(* Logix 5000 project; controller Receptivo vendor 1 type 14 code 106 rev 30.11; software revision 30.00 *)

TASK HARDWARE_TESTING (periodic, rate 67.76 ms, priority 7, watchdog 500 ms) : SYSTEM_STATUS
TASK MainTask (continuous, watchdog 500 ms) : MainProgram, Pesaje, Manejo_Productos, Calculo_Produccion

MODULES
   Local : vendor 1 type 14 code 106 (Compact 0, rev 30.11)
      Printer_Code_2D : vendor 1421 type 43 code 1000 (Ethernet 192.168.105.118, rev 1.1, StandardDataDriven RPI 100 ms)
           Printer_Code_2D:O.RawParserData[15]   // SLASH
           Printer_Code_2D:O.RawParserData[18]   // SLASH
           Printer_Code_2D:O.RawParserData[22]   // espacio
           Printer_Code_2D:O.RawParserData[129]   // campo 12
           Printer_Code_2D:O.RawParserData[23]   // ESPACIO
           Printer_Code_2D:O.RawParserData[27]   // minutos
           Printer_Code_2D:O.RawParserData[28]   // espacio
           Printer_Code_2D:O.RawParserData[36]   // operador
           Printer_Code_2D:O.RawParserData[19]   // year
           Printer_Code_2D:O.RawParserData[20]   // year
           Printer_Code_2D:O.RawParserData[34]   // CLIMA
           Printer_Code_2D:O.RawParserData[3]   // campo 11
           Printer_Code_2D:O.RawParserData[105]   // espacio
           Printer_Code_2D:O.RawParserData[29]   // ESPACIO
           Printer_Code_2D:O.RawParserData[37]   // OPERADOR
           Printer_Code_2D:O.RawParserData[33]   // ESPACIO
           Printer_Code_2D:O.RawParserData[113]   // PESO REAL
           Printer_Code_2D:O.RawParserData[26]   // DOS PUNTOS
           Printer_Code_2D:O.RawParserData[8]   // field data
           Printer_Code_2D:O.RawParserData[35]   // ESPACIO
           Printer_Code_2D:O.RawParserData[21]   // year
           Printer_Code_2D:O.RawParserData[24]   // hora
           Printer_Code_2D:O.RawParserData[25]   // HORA
           Printer_Code_2D:O.RawParserData[30]   // lote
           Printer_Code_2D:O.RawParserData[31]   // lote
           Printer_Code_2D:O.RawParserData[32]   // LOTE
           Printer_Code_2D:O.RawParserData[13]   // dia
           Printer_Code_2D:O.RawParserData[14]   // DIA
           Printer_Code_2D:O.RawParserData[16]   // mes
           Printer_Code_2D:O.RawParserData[17]   // MES
           Printer_Code_2D:O.RawParserData[10]   // codigo QR
           Printer_Code_2D:O.RawParserData[112]   // ESPACIO
           Printer_Code_2D:O.RawParserData[116]   // ESPACIO
           Printer_Code_2D:O.RawParserData[91]   // CODIGO EAN14
           Printer_Code_2D:O.RawParserData[38]   // ESPACIO
           Printer_Code_2D:O.RawParserData[90]   // ESPACIO
           Printer_Code_2D:O.RawParserData[106]   // CODIGO QAD 6 CARACTERES
           Printer_Code_2D:O.RawParserData[124]   // separador
           Printer_Code_2D:O.RawParserData[11]   // codigo QR
           Printer_Code_2D:O.RawParserData[120]   // ESPACIO
           Printer_Code_2D:O.RawParserData[121]   // NUMERO DE CAJAS
           Printer_Code_2D:O.RawParserData[12]   // codigo qr
           Printer_Code_2D:O.RawParserData[117]   // peso teorico
           Printer_Code_2D:O.RawParserData[39]   // DESCRIPCION
           Printer_Code_2D:O.RawParserData[127]   // nuevo campo
           Printer_Code_2D:O.RawParserData[132]   // field 12 data
           Printer_Code_2D:O.RawParserData[125]   // Numero Estacion
      Hardy_Basculas : vendor 258 type 43 code 3 (Ethernet 192.168.105.216, rev 2.37, StandardDataDriven RPI 100 ms)
END_MODULES

TYPE APT :
STRUCT
   Cod_QAD : DINT;
   Peso : DINT;
   Cajas : DINT;
END_STRUCT
END_TYPE

TYPE Codigo_Barras :
STRUCT
   LEN : DINT;
   DATA : SINT[14];
END_STRUCT
END_TYPE

TYPE Consecutivo :
STRUCT
   Consec : STRING[3];
END_STRUCT
END_TYPE

TYPE Descripcion :
STRUCT
   LEN : DINT;
   DATA : SINT[45];
END_STRUCT
END_TYPE

TYPE Ethernet_Status :
STRUCT
   EntryStatus : DINT[256];
   ConnStatus : INT[256];
   ConnFault : BOOL[256];
END_STRUCT
END_TYPE

TYPE Hora_y_Fecha :
STRUCT
   year : DINT;
   Mes : DINT;
   Dia : DINT;
   Hora : DINT;
   Minuto : DINT;
   Segundo : DINT;
   Milisegundos : DINT;
END_STRUCT
END_TYPE

TYPE MajorFaultBits :
STRUCT
   B_reserved : BOOL;
   B_PowerLoss : BOOL;
   B_reserved1 : BOOL;
   B_IO : BOOL;
   B_InstructionExecution : BOOL;
   B_FaultHandler : BOOL;
   B_Watchdog : BOOL;
   B_Stack : BOOL;
   B_ModeChange : BOOL;
   B_reserved2 : BOOL;
   B_reserved3 : BOOL;
   B_Motion : BOOL;
   B_reserved4 : BOOL;
   B_reserved5 : BOOL;
   B_reserved6 : BOOL;
   B_reserved7 : BOOL;
END_STRUCT
END_TYPE

TYPE MinorFaultBits :
STRUCT
   B_reserved1 : BOOL;
   B_reserved2 : BOOL;
   B_reserved3 : BOOL;
   B_reserved4 : BOOL;
   B_InstructionExecution : BOOL;
   B_reserved5 : BOOL;
   B_Watchdog : BOOL;
   B_reserved7 : BOOL;
   B_reserved8 : BOOL;
   B_SerialPort : BOOL;
   B_Battery : BOOL;
   B_reserved11 : BOOL;
   B_reserved12 : BOOL;
   B_reserved13 : BOOL;
   B_reserved14 : BOOL;
   B_reserved15 : BOOL;
END_STRUCT
END_TYPE

TYPE QR :
STRUCT
   LEN : DINT;
   DATA : SINT[112];
END_STRUCT
END_TYPE

TYPE Revision_Peso :
STRUCT
   Date : Hora_y_Fecha;
   Peso_Real : REAL;
   Peso_Teorico : REAL;
   Codigo : STRING;
END_STRUCT
END_TYPE

TYPE UDT_CAJAS :
STRUCT
   No_Cajas : STRING[2];
END_STRUCT
END_TYPE

TYPE UDT_COLA :
STRUCT
   Fecha : Hora_y_Fecha;
   Lote : INT;
   Operador : SINT;
   Descripcion : STRING;
   EAN14 : STRING;
   QAD : STRING;
   Peso_Real : REAL;
   Peso_Teorico : REAL;
   No_Cajas : INT;
   Clima : SINT;
   Consec : DINT;
   Envase : DINT;
   Envases_x_Caja : DINT;
   Peso_Insumos_Caja : REAL;
   Densidad_Medida : REAL;
   Linea : SINT;
END_STRUCT
END_TYPE

TYPE UDT_Densidad :
STRUCT
   Densidad : REAL;
   Fecha : Hora_y_Fecha;
END_STRUCT
END_TYPE

TYPE UDT_EAN14 :   // campo nuero dos del codigo QR
STRUCT
   EAN14 : STRING;
END_STRUCT
END_TYPE

TYPE UDT_GENERAL :
STRUCT
   dd : STRING[2];
   mm : STRING[2];
   yy : STRING[4];
   hh : STRING[2];
   min : STRING[2];
   lote : STRING[3];
   clima : STRING;
   operador : STRING[2];
   Descripcion : STRING;
   EAN14 : STRING;
   QAD : STRING;
   Peso_Real : STRING[3];
   Peso_Teorico : STRING[3];
   No_Cajas : STRING[3];
   Linea : STRING;
END_STRUCT
END_TYPE

TYPE UDT_Inventario :
STRUCT
   Peso_Real : REAL;
   Peso_Teorico_Caja : REAL;
   Peso_Teorico_Estiba : REAL;
   Codigo_EAN : STRING;
   Codigo_QAD : STRING;
   Codigo_Gco : STRING;
   Descripcion : Descripcion;
   CajaXEstiba : INT;
   Lote : INT;
   Clima : SINT;
   Linea : SINT;
   Codigo_Aceite : DINT;
END_STRUCT
END_TYPE

TYPE UDT_Maestro :
STRUCT
   Peso_Real_Estiba : REAL;
   Peso_Teorico_Caja : REAL;
   Codigo_EAN : STRING;
   Codigo_QAD : STRING;
   Codigo_GCO : DINT;
   Descripcion : STRING;
   Cajas_X_Estiba : DINT;
   Clima : DINT;
   Codigo_Aceite : DINT;
   Envase : DINT;
   Envases_x_Caja : DINT;
END_STRUCT
END_TYPE

TYPE UDT_PESO_REAL :   // quinto campo del codigo QR
STRUCT
   Peso_Real : STRING[2];
END_STRUCT
END_TYPE

TYPE UDT_PESO_TEORICO :   // sexto campo del codigo QR
STRUCT
   Peso_Teorico : STRING[2];
END_STRUCT
END_TYPE

TYPE UDT_Productos :   // Base de datos de Productos
STRUCT
   Peso_Real : REAL;
   Peso_Teorico_Caja : REAL;
   Codigo_EAN : Codigo_Barras;
   Codigo_QAD : DINT;
   Codigo_GCO : DINT;
   Cajas_x_Estiba : DINT;
   Clima : DINT;
   Descripcion : Descripcion;
END_STRUCT
END_TYPE

TYPE UDT_QAD :   // campo tres del codigo QR
STRUCT
   Codigo : STRING;
END_STRUCT
END_TYPE

TYPE WPM_Status :
STRUCT
   ADC_Error : BOOL;
   Reserved1 : BOOL;
   Not_Connected : BOOL;
   Over_Range : BOOL;
   Reserved2 : BOOL;
   Reserved3 : BOOL;
   In_Motion : BOOL;
   Firmware_Update : BOOL;
   Missing_Sample : BOOL;
   Channel_Off : BOOL;
   Failed_To_Save_To_Memory : BOOL;
   Update_In_Progress : BOOL;
   Failed_To_Update : BOOL;
   Saving_To_Memory : BOOL;
   It_Test_In_Progress : BOOL;
   Parameter_ID_Not_Found : BOOL;
   dato1 : INT;
END_STRUCT
END_TYPE

VAR_GLOBAL   (* controller tags *)
   ACTIVE_SLOT : DINT[10];
   Actualiza1_Timer : TIMER := (PRE := 7000);
   Actualiza2_Timer : TIMER := (PRE := 9000);
   Actualiza3_Timer : TIMER := (PRE := 6000);
   Actualiza4_Timer : TIMER := (PRE := 6000);
   Actualiza_Reporte_1 : BOOL;
   Actualiza_Reporte_2 : BOOL;
   Actualiza_Reporte_3 : BOOL;
   Actualiza_Reporte_4 : BOOL;
   ando : DINT := -1073741824;
   Ano_Biciesto : INT := 2020;
   Autonegotiation_Fallo : BOOL;
   Autonegotiation_OK : BOOL := 1;
   Autonegotiation_Start : BOOL;
   AutoNegotiation_Status : SINT := 3;
   Bit_Medianoche : BOOL;
   bit_ptobar : BOOL;
   CAJAS_1 : DINT := 50;
   CAJAS_2 : DINT := 56;
   CAJAS_3 : DINT := 50;
   CAJAS_4 : DINT := 48;
   Cajas_Aux : DINT;
   Cajas_Aux_Scanner : STRING;
   Cajas_Calculadas_Estacion_1 : REAL := -1.3294798;
   Cajas_Calculadas_Estacion_2 : REAL := -2.8708134;
   Cajas_Calculadas_Estacion_3 : REAL;
   Cajas_Calculadas_Estacion_4 : REAL := -1.4041514;
   Cajas_CalculadasG_Estacion_1 : REAL := 49.59538;
   Cajas_CalculadasG_Estacion_2 : REAL := 52.440193;
   Cajas_CalculadasG_Estacion_3 : REAL := 3.0057805;
   Cajas_CalculadasG_Estacion_4 : REAL := 48.046402;
   Calendario : Hora_y_Fecha := (year := 2021, Mes := 5, Dia := 28, Hora := 16, Minuto := 19, Segundo := 32, Milisegundos := 517635);
   Cant_total : SINT := 50;
   Cantidad_de_Productos : DINT := 117;
   CERO : DINT;
   CEROS : SINT;
   CHASSIS_LAST : DINT := 1;
   CINCO : SINT := 5;
   Clima_1 : DINT;
   Clima_2 : DINT;
   Clima_3 : DINT;
   Clima_4 : DINT;
   CLOCK : DINT[7] := ([0] := 2021, [1] := 5, [2] := 28, [3] := 16, [4] := 19, [5] := 33, [6] := 245632);
   codigo_capturado_1 : BOOL;
   codigo_capturado_2 : BOOL;
   codigo_capturado_3 : BOOL;
   codigo_capturado_4 : BOOL;
   Codigo_Encontrado : BOOL := 1;
   Codigo_QAD2_Espacios : DINT := 112;
   Cola_Densidad_Bidon_Ayer : REAL[50];
   Cola_Densidad_Bidon_Fecha_Ayer : Hora_y_Fecha[50];
   Cola_Densidad_Bidones : REAL[50];
   Cola_Densidad_Bidones_Fecha : Hora_y_Fecha[50];
   Cola_Densidad_Bidones_Fecha_Ayer : Hora_y_Fecha[50];
   Cola_Densidad_Elmar : REAL[50];
   Cola_Densidad_Elmar_Ayer : REAL[50];
   Cola_Densidad_Elmar_Fecha : Hora_y_Fecha[50];
   Cola_Densidad_Elmar_Fecha_Ayer : Hora_y_Fecha[50];
   Cola_Densidad_Fogg1 : REAL[50];
   Cola_Densidad_Fogg1_Ayer : REAL[50];
   Cola_Densidad_fogg1_Fecha : Hora_y_Fecha[50];
   Cola_Densidad_fogg1_Fecha_Ayer : Hora_y_Fecha[50];
   Cola_Densidad_Fogg2 : REAL[50];
   Cola_Densidad_Fogg2_Ayer : REAL[50];
   Cola_Densidad_fogg2_Fecha : Hora_y_Fecha[50];
   Cola_Densidad_fogg2_Fecha_Ayer : Hora_y_Fecha[50];
   Cola_Densidad_Karat : REAL[50];
   Cola_Densidad_Karat_Ayer : REAL[50];
   Cola_Densidad_Karat_Fecha : Hora_y_Fecha[50];
   Cola_Densidad_Karat_Fecha_Ayer : Hora_y_Fecha[50];
   Cola_Estacion_1 : UDT_COLA[100];
   Cola_Estacion_1_A : UDT_COLA[100];
   Cola_Estacion_2 : UDT_COLA[100] := ([0].Fecha.year := 2021, [0].Fecha.Mes := 5, [0].Fecha.Dia := 28, [0].Fecha.Hora := 11, [0].Fecha.Minuto := 23, [0].Fecha.Segundo := 35, [0].Fecha.Milisegundos := 472457, [0].Lote := 148, [0].Operador := 5, [0].Descripcion := 'Alegria Caja 12 x 900 cm3  - Costa', [0].EAN14 := '17702161409646', [0].QAD := '600620', [0].Peso_Real := 589.0, [0].Peso_Teorico := 585.0, [0].No_Cajas := 56, [0].Consec := 31, [0].Envase := 900, [0].Envases_x_Caja := 12, [0].Densidad_Medida := 0.9152, [0].Linea := 1, [1].Fecha.year := 2021, [1].Fecha.Mes := 5, [1].Fecha.Dia := 28, [1].Fecha.Hora := 11, [1].Fecha.Minuto := 26, [1].Fecha.Segundo := 22, [1].Fecha.Milisegundos := 21267, [1].Lote := 148, [1].Operador := 5, [1].Descripcion := 'Alegria Caja 12 x 900 cm3  - Costa', [1].EAN14 := '17702161409646', [1].QAD := '600620', [1].Peso_Real := 590.0, [1].Peso_Teorico := 585.0, [1].No_Cajas := 56, [1].Consec := 32, [1].Envase := 900, [1].Envases_x_Caja := 12, [1].Densidad_Medida := 0.9152, [1].Linea := 1, [2].Fecha.year := 2021, [2].Fecha.Mes := 5, [2].Fecha.Dia := 28, [2].Fecha.Hora := 11, [2].Fecha.Minuto := 29, [2].Fecha.Segundo := 36, [2].Fecha.Milisegundos := 993294, [2].Lote := 148, [2].Operador := 5, [2].Descripcion := 'Alegria Caja 12 x 900 cm3  - Costa', [2].EAN14 := '17702161409646', [2].QAD := '600620', [2].Peso_Real := 584.0, [2].Peso_Teorico := 585.0, [2].No_Cajas := 56, [2].Consec := 33, [2].Envase := 900, [2].Envases_x_Caja := 12, [2].Densidad_Medida := 0.9152, [2].Linea := 1,
        [3].Fecha.year := 2021, [3].Fecha.Mes := 5, [3].Fecha.Dia := 28, [3].Fecha.Hora := 11, [3].Fecha.Minuto := 32, [3].Fecha.Segundo := 47, [3].Fecha.Milisegundos := 567933, [3].Lote := 148, [3].Operador := 5, [3].Descripcion := 'Alegria Caja 12 x 900 cm3  - Costa', [3].EAN14 := '17702161409646', [3].QAD := '600620', [3].Peso_Real := 589.0, [3].Peso_Teorico := 585.0, [3].No_Cajas := 56, [3].Consec := 34, [3].Envase := 900, [3].Envases_x_Caja := 12, [3].Densidad_Medida := 0.9152, [3].Linea := 1, [4].Fecha.year := 2021, [4].Fecha.Mes := 5, [4].Fecha.Dia := 28, [4].Fecha.Hora := 11, [4].Fecha.Minuto := 35, [4].Fecha.Segundo := 25, [4].Fecha.Milisegundos := 115498, [4].Lote := 148, [4].Operador := 5, [4].Descripcion := 'Alegria Caja 12 x 900 cm3  - Costa', [4].EAN14 := '17702161409646', [4].QAD := '600620', [4].Peso_Real := 590.0, [4].Peso_Teorico := 585.0, [4].No_Cajas := 56, [4].Consec := 35, [4].Envase := 900, [4].Envases_x_Caja := 12, [4].Densidad_Medida := 0.9152, [4].Linea := 1, [5].Fecha.year := 2021, [5].Fecha.Mes := 5, [5].Fecha.Dia := 28, [5].Fecha.Hora := 11, [5].Fecha.Minuto := 38, [5].Fecha.Segundo := 2, [5].Fecha.Milisegundos := 738210, [5].Lote := 148, [5].Operador := 5, [5].Descripcion := 'Alegria Caja 12 x 900 cm3  - Costa', [5].EAN14 := '17702161409646', [5].QAD := '600620', [5].Peso_Real := 589.0, [5].Peso_Teorico := 585.0, [5].No_Cajas := 56, [5].Consec := 36, [5].Envase := 900, [5].Envases_x_Caja := 12, [5].Densidad_Medida := 0.9152, [5].Linea := 1,
        [6].Fecha.year := 2021, [6].Fecha.Mes := 5, [6].Fecha.Dia := 28, [6].Fecha.Hora := 11, [6].Fecha.Minuto := 40, [6].Fecha.Segundo := 46, [6].Fecha.Milisegundos := 866704, [6].Lote := 148, [6].Operador := 5, [6].Descripcion := 'Alegria Caja 12 x 900 cm3  - Costa', [6].EAN14 := '17702161409646', [6].QAD := '600620', [6].Peso_Real := 590.0, [6].Peso_Teorico := 585.0, [6].No_Cajas := 56, [6].Consec := 38, [6].Envase := 900, [6].Envases_x_Caja := 12, [6].Densidad_Medida := 0.9152, [6].Linea := 1, [7].Fecha.year := 2021, [7].Fecha.Mes := 5, [7].Fecha.Dia := 28, [7].Fecha.Hora := 11, [7].Fecha.Minuto := 44, [7].Fecha.Segundo := 7, [7].Fecha.Milisegundos := 219454, [7].Lote := 148, [7].Operador := 5, [7].Descripcion := 'Alegria Caja 12 x 900 cm3  - Costa', [7].EAN14 := '17702161409646', [7].QAD := '600620', [7].Peso_Real := 590.0, [7].Peso_Teorico := 585.0, [7].No_Cajas := 56, [7].Consec := 40, [7].Envase := 900, [7].Envases_x_Caja := 12, [7].Densidad_Medida := 0.9152, [7].Linea := 1, [8].Fecha.year := 2021, [8].Fecha.Mes := 5, [8].Fecha.Dia := 28, [8].Fecha.Hora := 11, [8].Fecha.Minuto := 46, [8].Fecha.Segundo := 55, [8].Fecha.Milisegundos := 872733, [8].Lote := 148, [8].Operador := 5, [8].Descripcion := 'Alegria Caja 12 x 900 cm3  - Costa', [8].EAN14 := '17702161409646', [8].QAD := '600620', [8].Peso_Real := 590.0, [8].Peso_Teorico := 585.0, [8].No_Cajas := 56, [8].Consec := 41, [8].Envase := 900, [8].Envases_x_Caja := 12, [8].Densidad_Medida := 0.9152, [8].Linea := 1,
        [9].Fecha.year := 2021, [9].Fecha.Mes := 5, [9].Fecha.Dia := 28, [9].Fecha.Hora := 11, [9].Fecha.Minuto := 49, [9].Fecha.Segundo := 6, [9].Fecha.Milisegundos := 938412, [9].Lote := 148, [9].Operador := 5, [9].Descripcion := 'Alegria Caja 12 x 900 cm3  - Costa', [9].EAN14 := '17702161409646', [9].QAD := '600620', [9].Peso_Real := 590.0, [9].Peso_Teorico := 585.0, [9].No_Cajas := 56, [9].Consec := 43, [9].Envase := 900, [9].Envases_x_Caja := 12, [9].Densidad_Medida := 0.9152, [9].Linea := 1, [10].Fecha.year := 2021, [10].Fecha.Mes := 5, [10].Fecha.Dia := 28, [10].Fecha.Hora := 11, [10].Fecha.Minuto := 51, [10].Fecha.Segundo := 47, [10].Fecha.Milisegundos := 512506, [10].Lote := 148, [10].Operador := 5, [10].Descripcion := 'Alegria Caja 12 x 900 cm3  - Costa', [10].EAN14 := '17702161409646', [10].QAD := '600620', [10].Peso_Real := 590.0, [10].Peso_Teorico := 585.0, [10].No_Cajas := 56, [10].Consec := 44, [10].Envase := 900, [10].Envases_x_Caja := 12, [10].Densidad_Medida := 0.9152, [10].Linea := 1, [11].Fecha.year := 2021, [11].Fecha.Mes := 5, [11].Fecha.Dia := 28, [11].Fecha.Hora := 11, [11].Fecha.Minuto := 54, [11].Fecha.Segundo := 6, [11].Fecha.Milisegundos := 98780, [11].Lote := 148, [11].Operador := 5, [11].Descripcion := 'Alegria Caja 12 x 900 cm3  - Costa', [11].EAN14 := '17702161409646', [11].QAD := '600620', [11].Peso_Real := 590.0, [11].Peso_Teorico := 585.0, [11].No_Cajas := 56, [11].Consec := 45, [11].Envase := 900, [11].Envases_x_Caja := 12, [11].Densidad_Medida := 0.9152, [11].Linea := 1,
        [12].Fecha.year := 2021, [12].Fecha.Mes := 5, [12].Fecha.Dia := 28, [12].Fecha.Hora := 11, [12].Fecha.Minuto := 56, [12].Fecha.Segundo := 16, [12].Fecha.Milisegundos := 868293, [12].Lote := 148, [12].Operador := 5, [12].Descripcion := 'Alegria Caja 12 x 900 cm3  - Costa', [12].EAN14 := '17702161409646', [12].QAD := '600620', [12].Peso_Real := 591.0, [12].Peso_Teorico := 585.0, [12].No_Cajas := 56, [12].Consec := 47, [12].Envase := 900, [12].Envases_x_Caja := 12, [12].Densidad_Medida := 0.9152, [12].Linea := 1, [13].Fecha.year := 2021, [13].Fecha.Mes := 5, [13].Fecha.Dia := 28, [13].Fecha.Hora := 11, [13].Fecha.Minuto := 58, [13].Fecha.Segundo := 33, [13].Fecha.Milisegundos := 275353, [13].Lote := 148, [13].Operador := 5, [13].Descripcion := 'Alegria Caja 12 x 900 cm3  - Costa', [13].EAN14 := '17702161409646', [13].QAD := '600620', [13].Peso_Real := 591.0, [13].Peso_Teorico := 585.0, [13].No_Cajas := 56, [13].Consec := 48, [13].Envase := 900, [13].Envases_x_Caja := 12, [13].Densidad_Medida := 0.9152, [13].Linea := 1, [14].Fecha.year := 2021, [14].Fecha.Mes := 5, [14].Fecha.Dia := 28, [14].Fecha.Hora := 12, [14].Fecha.Segundo := 51, [14].Fecha.Milisegundos := 241323, [14].Lote := 148, [14].Operador := 5, [14].Descripcion := 'Alegria Caja 12 x 900 cm3  - Costa', [14].EAN14 := '17702161409646', [14].QAD := '600620', [14].Peso_Real := 590.0, [14].Peso_Teorico := 585.0, [14].No_Cajas := 56, [14].Consec := 49, [14].Envase := 900, [14].Envases_x_Caja := 12, [14].Densidad_Medida := 0.9152, [14].Linea := 1, [15].Fecha.year := 2021,
        [15].Fecha.Mes := 5, [15].Fecha.Dia := 28, [15].Fecha.Hora := 12, [15].Fecha.Minuto := 3, [15].Fecha.Segundo := 25, [15].Fecha.Milisegundos := 977302, [15].Lote := 148, [15].Operador := 5, [15].Descripcion := 'Alegria Caja 12 x 900 cm3  - Costa', [15].EAN14 := '17702161409646', [15].QAD := '600620', [15].Peso_Real := 589.0, [15].Peso_Teorico := 585.0, [15].No_Cajas := 56, [15].Consec := 50, [15].Envase := 900, [15].Envases_x_Caja := 12, [15].Densidad_Medida := 0.9152, [15].Linea := 1, [16].Fecha.year := 2021, [16].Fecha.Mes := 5, [16].Fecha.Dia := 28, [16].Fecha.Hora := 12, [16].Fecha.Minuto := 5, [16].Fecha.Segundo := 59, [16].Fecha.Milisegundos := 211755, [16].Lote := 148, [16].Operador := 5, [16].Descripcion := 'Alegria Caja 12 x 900 cm3  - Costa', [16].EAN14 := '17702161409646', [16].QAD := '600620', [16].Peso_Real := 589.0, [16].Peso_Teorico := 585.0, [16].No_Cajas := 56, [16].Consec := 51, [16].Envase := 900, [16].Envases_x_Caja := 12, [16].Densidad_Medida := 0.9152, [16].Linea := 1, [17].Fecha.year := 2021, [17].Fecha.Mes := 5, [17].Fecha.Dia := 28, [17].Fecha.Hora := 12, [17].Fecha.Minuto := 8, [17].Fecha.Segundo := 18, [17].Fecha.Milisegundos := 641820, [17].Lote := 148, [17].Operador := 5, [17].Descripcion := 'Alegria Caja 12 x 900 cm3  - Costa', [17].EAN14 := '17702161409646', [17].QAD := '600620', [17].Peso_Real := 589.0, [17].Peso_Teorico := 585.0, [17].No_Cajas := 56, [17].Consec := 52, [17].Envase := 900, [17].Envases_x_Caja := 12, [17].Densidad_Medida := 0.9152, [17].Linea := 1, [18].Fecha.year := 2021,
        [18].Fecha.Mes := 5, [18].Fecha.Dia := 28, [18].Fecha.Hora := 12, [18].Fecha.Minuto := 10, [18].Fecha.Segundo := 49, [18].Fecha.Milisegundos := 898961, [18].Lote := 148, [18].Operador := 5, [18].Descripcion := 'Alegria Caja 12 x 900 cm3  - Costa', [18].EAN14 := '17702161409646', [18].QAD := '600620', [18].Peso_Real := 589.0, [18].Peso_Teorico := 585.0, [18].No_Cajas := 56, [18].Consec := 53, [18].Envase := 900, [18].Envases_x_Caja := 12, [18].Densidad_Medida := 0.9152, [18].Linea := 1, [19].Fecha.year := 2021, [19].Fecha.Mes := 5, [19].Fecha.Dia := 28, [19].Fecha.Hora := 12, [19].Fecha.Minuto := 12, [19].Fecha.Segundo := 58, [19].Fecha.Milisegundos := 826984, [19].Lote := 148, [19].Operador := 5, [19].Descripcion := 'Alegria Caja 12 x 900 cm3  - Costa', [19].EAN14 := '17702161409646', [19].QAD := '600620', [19].Peso_Real := 589.0, [19].Peso_Teorico := 585.0, [19].No_Cajas := 56, [19].Consec := 54, [19].Envase := 900, [19].Envases_x_Caja := 12, [19].Densidad_Medida := 0.9152, [19].Linea := 1, [20].Fecha.year := 2021, [20].Fecha.Mes := 5, [20].Fecha.Dia := 28, [20].Fecha.Hora := 12, [20].Fecha.Minuto := 15, [20].Fecha.Segundo := 28, [20].Fecha.Milisegundos := 245825, [20].Lote := 148, [20].Operador := 5, [20].Descripcion := 'Alegria Caja 12 x 900 cm3  - Costa', [20].EAN14 := '17702161409646', [20].QAD := '600620', [20].Peso_Real := 588.0, [20].Peso_Teorico := 585.0, [20].No_Cajas := 56, [20].Consec := 55, [20].Envase := 900, [20].Envases_x_Caja := 12, [20].Densidad_Medida := 0.9152, [20].Linea := 1, [21].Fecha.year := 2021,
        [21].Fecha.Mes := 5, [21].Fecha.Dia := 28, [21].Fecha.Hora := 12, [21].Fecha.Minuto := 17, [21].Fecha.Segundo := 41, [21].Fecha.Milisegundos := 646158, [21].Lote := 148, [21].Operador := 5, [21].Descripcion := 'Alegria Caja 12 x 900 cm3  - Costa', [21].EAN14 := '17702161409646', [21].QAD := '600620', [21].Peso_Real := 589.0, [21].Peso_Teorico := 585.0, [21].No_Cajas := 56, [21].Consec := 56, [21].Envase := 900, [21].Envases_x_Caja := 12, [21].Densidad_Medida := 0.9152, [21].Linea := 1, [22].Fecha.year := 2021, [22].Fecha.Mes := 5, [22].Fecha.Dia := 28, [22].Fecha.Hora := 12, [22].Fecha.Minuto := 20, [22].Fecha.Segundo := 40, [22].Fecha.Milisegundos := 210367, [22].Lote := 148, [22].Operador := 5, [22].Descripcion := 'Alegria Caja 12 x 900 cm3  - Costa', [22].EAN14 := '17702161409646', [22].QAD := '600620', [22].Peso_Real := 588.0, [22].Peso_Teorico := 585.0, [22].No_Cajas := 56, [22].Consec := 57, [22].Envase := 900, [22].Envases_x_Caja := 12, [22].Densidad_Medida := 0.9152, [22].Linea := 1, [23].Fecha.year := 2021, [23].Fecha.Mes := 5, [23].Fecha.Dia := 28, [23].Fecha.Hora := 12, [23].Fecha.Minuto := 22, [23].Fecha.Segundo := 35, [23].Fecha.Milisegundos := 762553, [23].Lote := 148, [23].Operador := 5, [23].Descripcion := 'Alegria Caja 12 x 900 cm3  - Costa', [23].EAN14 := '17702161409646', [23].QAD := '600620', [23].Peso_Real := 590.0, [23].Peso_Teorico := 585.0, [23].No_Cajas := 56, [23].Consec := 58, [23].Envase := 900, [23].Envases_x_Caja := 12, [23].Densidad_Medida := 0.9152, [23].Linea := 1, [24].Fecha.year := 2021,
        [24].Fecha.Mes := 5, [24].Fecha.Dia := 28, [24].Fecha.Hora := 12, [24].Fecha.Minuto := 29, [24].Fecha.Segundo := 23, [24].Fecha.Milisegundos := 722342, [24].Lote := 148, [24].Operador := 5, [24].Descripcion := 'Alegria Caja 12 x 900 cm3  - Costa', [24].EAN14 := '17702161409646', [24].QAD := '600620', [24].Peso_Real := 587.0, [24].Peso_Teorico := 585.0, [24].No_Cajas := 56, [24].Consec := 59, [24].Envase := 900, [24].Envases_x_Caja := 12, [24].Densidad_Medida := 0.9152, [24].Linea := 1, [25].Fecha.year := 2021, [25].Fecha.Mes := 5, [25].Fecha.Dia := 28, [25].Fecha.Hora := 12, [25].Fecha.Minuto := 36, [25].Fecha.Segundo := 23, [25].Fecha.Milisegundos := 316720, [25].Lote := 148, [25].Operador := 5, [25].Descripcion := 'Alegria Caja 12 x 900 cm3  - Costa', [25].EAN14 := '17702161409646', [25].QAD := '600620', [25].Peso_Real := 586.0, [25].Peso_Teorico := 585.0, [25].No_Cajas := 56, [25].Consec := 60, [25].Envase := 900, [25].Envases_x_Caja := 12, [25].Densidad_Medida := 0.9152, [25].Linea := 1, [26].Fecha.year := 2021, [26].Fecha.Mes := 5, [26].Fecha.Dia := 28, [26].Fecha.Hora := 12, [26].Fecha.Minuto := 38, [26].Fecha.Segundo := 23, [26].Fecha.Milisegundos := 44403, [26].Lote := 148, [26].Operador := 5, [26].Descripcion := 'Alegria Caja 12 x 900 cm3  - Costa', [26].EAN14 := '17702161409646', [26].QAD := '600620', [26].Peso_Real := 579.0, [26].Peso_Teorico := 585.0, [26].No_Cajas := 56, [26].Consec := 62, [26].Envase := 900, [26].Envases_x_Caja := 12, [26].Densidad_Medida := 0.9152, [26].Linea := 1, [27].Fecha.year := 2021,
        [27].Fecha.Mes := 5, [27].Fecha.Dia := 28, [27].Fecha.Hora := 12, [27].Fecha.Minuto := 47, [27].Fecha.Segundo := 26, [27].Fecha.Milisegundos := 654204, [27].Lote := 148, [27].Operador := 5, [27].Descripcion := 'Alegria Caja 12 x 900 cm3  - Costa', [27].EAN14 := '17702161409646', [27].QAD := '600620', [27].Peso_Real := 578.0, [27].Peso_Teorico := 585.0, [27].No_Cajas := 56, [27].Consec := 63, [27].Envase := 900, [27].Envases_x_Caja := 12, [27].Densidad_Medida := 0.9152, [27].Linea := 1, [28].Fecha.year := 2021, [28].Fecha.Mes := 5, [28].Fecha.Dia := 28, [28].Fecha.Hora := 12, [28].Fecha.Minuto := 50, [28].Fecha.Segundo := 58, [28].Fecha.Milisegundos := 76476, [28].Lote := 148, [28].Operador := 5, [28].Descripcion := 'Alegria Caja 12 x 900 cm3  - Costa', [28].EAN14 := '17702161409646', [28].QAD := '600620', [28].Peso_Real := 602.0, [28].Peso_Teorico := 585.0, [28].No_Cajas := 56, [28].Consec := 65, [28].Envase := 900, [28].Envases_x_Caja := 12, [28].Densidad_Medida := 0.9152, [28].Linea := 1, [29].Fecha.year := 2021, [29].Fecha.Mes := 5, [29].Fecha.Dia := 28, [29].Fecha.Hora := 12, [29].Fecha.Minuto := 53, [29].Fecha.Segundo := 51, [29].Fecha.Milisegundos := 99875, [29].Lote := 148, [29].Operador := 5, [29].Descripcion := 'Alegria Caja 12 x 900 cm3  - Costa', [29].EAN14 := '17702161409646', [29].QAD := '600620', [29].Peso_Real := 592.0, [29].Peso_Teorico := 585.0, [29].No_Cajas := 56, [29].Consec := 67, [29].Envase := 900, [29].Envases_x_Caja := 12, [29].Densidad_Medida := 0.9152, [29].Linea := 1, [30].Fecha.year := 2021,
        [30].Fecha.Mes := 5, [30].Fecha.Dia := 28, [30].Fecha.Hora := 13, [30].Fecha.Minuto := 3, [30].Fecha.Segundo := 33, [30].Fecha.Milisegundos := 200046, [30].Lote := 148, [30].Operador := 5, [30].Descripcion := 'Alegria Caja 12 x 900 cm3  - Costa', [30].EAN14 := '17702161409646', [30].QAD := '600620', [30].Peso_Real := 588.0, [30].Peso_Teorico := 585.0, [30].No_Cajas := 56, [30].Consec := 69, [30].Envase := 900, [30].Envases_x_Caja := 12, [30].Densidad_Medida := 0.9152, [30].Linea := 1, [31].Fecha.year := 2021, [31].Fecha.Mes := 5, [31].Fecha.Dia := 28, [31].Fecha.Hora := 13, [31].Fecha.Minuto := 6, [31].Fecha.Segundo := 3, [31].Fecha.Milisegundos := 885977, [31].Lote := 148, [31].Operador := 5, [31].Descripcion := 'Alegria Caja 12 x 900 cm3  - Costa', [31].EAN14 := '17702161409646', [31].QAD := '600620', [31].Peso_Real := 590.0, [31].Peso_Teorico := 585.0, [31].No_Cajas := 56, [31].Consec := 71, [31].Envase := 900, [31].Envases_x_Caja := 12, [31].Densidad_Medida := 0.9152, [31].Linea := 1, [32].Fecha.year := 2021, [32].Fecha.Mes := 5, [32].Fecha.Dia := 28, [32].Fecha.Hora := 13, [32].Fecha.Minuto := 8, [32].Fecha.Segundo := 15, [32].Fecha.Milisegundos := 424465, [32].Lote := 148, [32].Operador := 5, [32].Descripcion := 'Alegria Caja 12 x 900 cm3  - Costa', [32].EAN14 := '17702161409646', [32].QAD := '600620', [32].Peso_Real := 592.0, [32].Peso_Teorico := 585.0, [32].No_Cajas := 56, [32].Consec := 72, [32].Envase := 900, [32].Envases_x_Caja := 12, [32].Densidad_Medida := 0.9152, [32].Linea := 1, [33].Fecha.year := 2021,
        [33].Fecha.Mes := 5, [33].Fecha.Dia := 28, [33].Fecha.Hora := 13, [33].Fecha.Minuto := 11, [33].Fecha.Segundo := 2, [33].Fecha.Milisegundos := 161258, [33].Lote := 148, [33].Operador := 5, [33].Descripcion := 'Alegria Caja 12 x 900 cm3  - Costa', [33].EAN14 := '17702161409646', [33].QAD := '600620', [33].Peso_Real := 586.0, [33].Peso_Teorico := 585.0, [33].No_Cajas := 56, [33].Consec := 74, [33].Envase := 900, [33].Envases_x_Caja := 12, [33].Densidad_Medida := 0.9152, [33].Linea := 1, [34].Fecha.year := 2021, [34].Fecha.Mes := 5, [34].Fecha.Dia := 28, [34].Fecha.Hora := 13, [34].Fecha.Minuto := 13, [34].Fecha.Segundo := 15, [34].Fecha.Milisegundos := 997430, [34].Lote := 148, [34].Operador := 5, [34].Descripcion := 'Alegria Caja 12 x 900 cm3  - Costa', [34].EAN14 := '17702161409646', [34].QAD := '600620', [34].Peso_Real := 595.0, [34].Peso_Teorico := 585.0, [34].No_Cajas := 56, [34].Consec := 75, [34].Envase := 900, [34].Envases_x_Caja := 12, [34].Densidad_Medida := 0.9152, [34].Linea := 1, [35].Fecha.year := 2021, [35].Fecha.Mes := 5, [35].Fecha.Dia := 28, [35].Fecha.Hora := 13, [35].Fecha.Minuto := 16, [35].Fecha.Segundo := 17, [35].Fecha.Milisegundos := 510044, [35].Lote := 148, [35].Operador := 5, [35].Descripcion := 'Alegria Caja 12 x 900 cm3  - Costa', [35].EAN14 := '17702161409646', [35].QAD := '600620', [35].Peso_Real := 592.0, [35].Peso_Teorico := 585.0, [35].No_Cajas := 56, [35].Consec := 76, [35].Envase := 900, [35].Envases_x_Caja := 12, [35].Densidad_Medida := 0.9152, [35].Linea := 1, [36].Fecha.year := 2021,
        [36].Fecha.Mes := 5, [36].Fecha.Dia := 28, [36].Fecha.Hora := 13, [36].Fecha.Minuto := 18, [36].Fecha.Segundo := 9, [36].Fecha.Milisegundos := 744490, [36].Lote := 148, [36].Operador := 5, [36].Descripcion := 'Alegria Caja 12 x 900 cm3  - Costa', [36].EAN14 := '17702161409646', [36].QAD := '600620', [36].Peso_Real := 592.0, [36].Peso_Teorico := 585.0, [36].No_Cajas := 56, [36].Consec := 77, [36].Envase := 900, [36].Envases_x_Caja := 12, [36].Densidad_Medida := 0.9152, [36].Linea := 1, [37].Fecha.year := 2021, [37].Fecha.Mes := 5, [37].Fecha.Dia := 28, [37].Fecha.Hora := 13, [37].Fecha.Minuto := 20, [37].Fecha.Segundo := 36, [37].Fecha.Milisegundos := 982435, [37].Lote := 148, [37].Operador := 5, [37].Descripcion := 'Alegria Caja 12 x 900 cm3  - Costa', [37].EAN14 := '17702161409646', [37].QAD := '600620', [37].Peso_Real := 592.0, [37].Peso_Teorico := 585.0, [37].No_Cajas := 56, [37].Consec := 79, [37].Envase := 900, [37].Envases_x_Caja := 12, [37].Densidad_Medida := 0.9152, [37].Linea := 1, [38].Fecha.year := 2021, [38].Fecha.Mes := 5, [38].Fecha.Dia := 28, [38].Fecha.Hora := 13, [38].Fecha.Minuto := 23, [38].Fecha.Segundo := 7, [38].Fecha.Milisegundos := 303111, [38].Lote := 148, [38].Operador := 5, [38].Descripcion := 'Alegria Caja 12 x 900 cm3  - Costa', [38].EAN14 := '17702161409646', [38].QAD := '600620', [38].Peso_Real := 592.0, [38].Peso_Teorico := 585.0, [38].No_Cajas := 56, [38].Consec := 80, [38].Envase := 900, [38].Envases_x_Caja := 12, [38].Densidad_Medida := 0.9152, [38].Linea := 1, [39].Fecha.year := 2021,
        [39].Fecha.Mes := 5, [39].Fecha.Dia := 28, [39].Fecha.Hora := 13, [39].Fecha.Minuto := 25, [39].Fecha.Segundo := 31, [39].Fecha.Milisegundos := 853442, [39].Lote := 148, [39].Operador := 5, [39].Descripcion := 'Alegria Caja 12 x 900 cm3  - Costa', [39].EAN14 := '17702161409646', [39].QAD := '600620', [39].Peso_Real := 592.0, [39].Peso_Teorico := 585.0, [39].No_Cajas := 56, [39].Consec := 82, [39].Envase := 900, [39].Envases_x_Caja := 12, [39].Densidad_Medida := 0.9152, [39].Linea := 1, [40].Fecha.year := 2021, [40].Fecha.Mes := 5, [40].Fecha.Dia := 28, [40].Fecha.Hora := 13, [40].Fecha.Minuto := 27, [40].Fecha.Segundo := 55, [40].Fecha.Milisegundos := 335071, [40].Lote := 148, [40].Operador := 5, [40].Descripcion := 'Alegria Caja 12 x 900 cm3  - Costa', [40].EAN14 := '17702161409646', [40].QAD := '600620', [40].Peso_Real := 588.0, [40].Peso_Teorico := 585.0, [40].No_Cajas := 56, [40].Consec := 83, [40].Envase := 900, [40].Envases_x_Caja := 12, [40].Densidad_Medida := 0.9152, [40].Linea := 1, [41].Fecha.year := 2021, [41].Fecha.Mes := 5, [41].Fecha.Dia := 28, [41].Fecha.Hora := 13, [41].Fecha.Minuto := 32, [41].Fecha.Segundo := 52, [41].Fecha.Milisegundos := 125206, [41].Lote := 148, [41].Operador := 5, [41].Descripcion := 'Alegria Caja 12 x 900 cm3  - Costa', [41].EAN14 := '17702161409646', [41].QAD := '600620', [41].Peso_Real := 592.0, [41].Peso_Teorico := 585.0, [41].No_Cajas := 56, [41].Consec := 85, [41].Envase := 900, [41].Envases_x_Caja := 12, [41].Densidad_Medida := 0.9152, [41].Linea := 1, [42].Fecha.year := 2021,
        [42].Fecha.Mes := 5, [42].Fecha.Dia := 28, [42].Fecha.Hora := 13, [42].Fecha.Minuto := 33, [42].Fecha.Segundo := 31, [42].Fecha.Milisegundos := 629888, [42].Lote := 148, [42].Operador := 5, [42].Descripcion := 'Alegria Caja 12 x 900 cm3  - Costa', [42].EAN14 := '17702161409646', [42].QAD := '600620', [42].Peso_Real := 593.0, [42].Peso_Teorico := 585.0, [42].No_Cajas := 56, [42].Consec := 86, [42].Envase := 900, [42].Envases_x_Caja := 12, [42].Densidad_Medida := 0.9152, [42].Linea := 1, [43].Fecha.year := 2021, [43].Fecha.Mes := 5, [43].Fecha.Dia := 28, [43].Fecha.Hora := 13, [43].Fecha.Minuto := 53, [43].Fecha.Segundo := 16, [43].Fecha.Milisegundos := 819629, [43].Lote := 148, [43].Operador := 5, [43].Descripcion := 'Alegria Caja 12 x 900 cm3  - Costa', [43].EAN14 := '17702161409646', [43].QAD := '600620', [43].Peso_Real := 591.0, [43].Peso_Teorico := 585.0, [43].No_Cajas := 56, [43].Consec := 89, [43].Envase := 900, [43].Envases_x_Caja := 12, [43].Densidad_Medida := 0.9152, [43].Linea := 1, [44].Fecha.year := 2021, [44].Fecha.Mes := 5, [44].Fecha.Dia := 28, [44].Fecha.Hora := 13, [44].Fecha.Minuto := 55, [44].Fecha.Segundo := 32, [44].Fecha.Milisegundos := 634598, [44].Lote := 148, [44].Operador := 5, [44].Descripcion := 'Alegria Caja 12 x 900 cm3  - Costa', [44].EAN14 := '17702161409646', [44].QAD := '600620', [44].Peso_Real := 592.0, [44].Peso_Teorico := 585.0, [44].No_Cajas := 56, [44].Consec := 91, [44].Envase := 900, [44].Envases_x_Caja := 12, [44].Densidad_Medida := 0.9152, [44].Linea := 1, [45].Fecha.year := 2021,
        [45].Fecha.Mes := 5, [45].Fecha.Dia := 28, [45].Fecha.Hora := 13, [45].Fecha.Minuto := 58, [45].Fecha.Segundo := 2, [45].Fecha.Milisegundos := 400890, [45].Lote := 148, [45].Operador := 5, [45].Descripcion := 'Alegria Caja 12 x 900 cm3  - Costa', [45].EAN14 := '17702161409646', [45].QAD := '600620', [45].Peso_Real := 592.0, [45].Peso_Teorico := 585.0, [45].No_Cajas := 56, [45].Consec := 92, [45].Envase := 900, [45].Envases_x_Caja := 12, [45].Densidad_Medida := 0.9152, [45].Linea := 1, [46].Fecha.year := 2021, [46].Fecha.Mes := 5, [46].Fecha.Dia := 28, [46].Fecha.Hora := 14, [46].Fecha.Segundo := 29, [46].Fecha.Milisegundos := 455405, [46].Lote := 148, [46].Operador := 5, [46].Descripcion := 'Alegria Caja 12 x 900 cm3  - Costa', [46].EAN14 := '17702161409646', [46].QAD := '600620', [46].Peso_Real := 584.0, [46].Peso_Teorico := 585.0, [46].No_Cajas := 56, [46].Consec := 93, [46].Envase := 900, [46].Envases_x_Caja := 12, [46].Densidad_Medida := 0.9152, [46].Linea := 1, [47].Fecha.year := 2021, [47].Fecha.Mes := 5, [47].Fecha.Dia := 28, [47].Fecha.Hora := 14, [47].Fecha.Minuto := 7, [47].Fecha.Segundo := 12, [47].Fecha.Milisegundos := 746049, [47].Lote := 148, [47].Operador := 5, [47].Descripcion := 'Alegria Caja 12 x 900 cm3  - Costa', [47].EAN14 := '17702161409646', [47].QAD := '600620', [47].Peso_Real := 592.0, [47].Peso_Teorico := 585.0, [47].No_Cajas := 56, [47].Consec := 95, [47].Envase := 900, [47].Envases_x_Caja := 12, [47].Densidad_Medida := 0.9152, [47].Linea := 1, [48].Fecha.year := 2021, [48].Fecha.Mes := 5,
        [48].Fecha.Dia := 28, [48].Fecha.Hora := 14, [48].Fecha.Minuto := 9, [48].Fecha.Segundo := 35, [48].Fecha.Milisegundos := 430366, [48].Lote := 148, [48].Operador := 5, [48].Descripcion := 'Alegria Caja 12 x 900 cm3  - Costa', [48].EAN14 := '17702161409646', [48].QAD := '600620', [48].Peso_Real := 590.0, [48].Peso_Teorico := 585.0, [48].No_Cajas := 56, [48].Consec := 96, [48].Envase := 900, [48].Envases_x_Caja := 12, [48].Densidad_Medida := 0.9152, [48].Linea := 1, [49].Fecha.year := 2021, [49].Fecha.Mes := 5, [49].Fecha.Dia := 28, [49].Fecha.Hora := 14, [49].Fecha.Minuto := 11, [49].Fecha.Segundo := 51, [49].Fecha.Milisegundos := 729293, [49].Lote := 148, [49].Operador := 5, [49].Descripcion := 'Alegria Caja 12 x 900 cm3  - Costa', [49].EAN14 := '17702161409646', [49].QAD := '600620', [49].Peso_Real := 589.0, [49].Peso_Teorico := 585.0, [49].No_Cajas := 56, [49].Consec := 97, [49].Envase := 900, [49].Envases_x_Caja := 12, [49].Densidad_Medida := 0.9152, [49].Linea := 1, [50].Fecha.year := 2021, [50].Fecha.Mes := 5, [50].Fecha.Dia := 28, [50].Fecha.Hora := 14, [50].Fecha.Minuto := 14, [50].Fecha.Segundo := 44, [50].Fecha.Milisegundos := 672944, [50].Lote := 148, [50].Operador := 5, [50].Descripcion := 'Alegria Caja 12 x 900 cm3  - Costa', [50].EAN14 := '17702161409646', [50].QAD := '600620', [50].Peso_Real := 590.0, [50].Peso_Teorico := 585.0, [50].No_Cajas := 56, [50].Consec := 99, [50].Envase := 900, [50].Envases_x_Caja := 12, [50].Densidad_Medida := 0.9152, [50].Linea := 1, [51].Fecha.year := 2021, [51].Fecha.Mes := 5,
        [51].Fecha.Dia := 28, [51].Fecha.Hora := 14, [51].Fecha.Minuto := 17, [51].Fecha.Segundo := 36, [51].Fecha.Milisegundos := 109035, [51].Lote := 148, [51].Operador := 5, [51].Descripcion := 'Alegria Caja 12 x 900 cm3  - Costa', [51].EAN14 := '17702161409646', [51].QAD := '600620', [51].Peso_Real := 591.0, [51].Peso_Teorico := 585.0, [51].No_Cajas := 56, [51].Consec := 100, [51].Envase := 900, [51].Envases_x_Caja := 12, [51].Densidad_Medida := 0.9152, [51].Linea := 1, [52].Fecha.year := 2021, [52].Fecha.Mes := 5, [52].Fecha.Dia := 28, [52].Fecha.Hora := 14, [52].Fecha.Minuto := 19, [52].Fecha.Segundo := 47, [52].Fecha.Milisegundos := 596775, [52].Lote := 148, [52].Operador := 5, [52].Descripcion := 'Alegria Caja 12 x 900 cm3  - Costa', [52].EAN14 := '17702161409646', [52].QAD := '600620', [52].Peso_Real := 592.0, [52].Peso_Teorico := 585.0, [52].No_Cajas := 56, [52].Consec := 101, [52].Envase := 900, [52].Envases_x_Caja := 12, [52].Densidad_Medida := 0.9152, [52].Linea := 1, [53].Fecha.year := 2021, [53].Fecha.Mes := 5, [53].Fecha.Dia := 28, [53].Fecha.Hora := 14, [53].Fecha.Minuto := 28, [53].Fecha.Segundo := 31, [53].Fecha.Milisegundos := 494425, [53].Lote := 148, [53].Operador := 5, [53].Descripcion := 'Alegria Caja 12 x 900 cm3  - Costa', [53].EAN14 := '17702161409646', [53].QAD := '600620', [53].Peso_Real := 591.0, [53].Peso_Teorico := 585.0, [53].No_Cajas := 56, [53].Consec := 104, [53].Envase := 900, [53].Envases_x_Caja := 12, [53].Densidad_Medida := 0.9152, [53].Linea := 1, [54].Fecha.year := 2021, [54].Fecha.Mes := 5,
        [54].Fecha.Dia := 28, [54].Fecha.Hora := 14, [54].Fecha.Minuto := 31, [54].Fecha.Segundo := 15, [54].Fecha.Milisegundos := 401683, [54].Lote := 148, [54].Operador := 5, [54].Descripcion := 'Alegria Caja 12 x 900 cm3  - Costa', [54].EAN14 := '17702161409646', [54].QAD := '600620', [54].Peso_Real := 587.0, [54].Peso_Teorico := 585.0, [54].No_Cajas := 56, [54].Consec := 105, [54].Envase := 900, [54].Envases_x_Caja := 12, [54].Densidad_Medida := 0.9152, [54].Linea := 1, [55].Fecha.year := 2021, [55].Fecha.Mes := 5, [55].Fecha.Dia := 28, [55].Fecha.Hora := 14, [55].Fecha.Minuto := 38, [55].Fecha.Segundo := 5, [55].Fecha.Milisegundos := 319333, [55].Lote := 148, [55].Operador := 5, [55].Descripcion := 'Alegria Caja 12 x 900 cm3  - Costa', [55].EAN14 := '17702161409646', [55].QAD := '600620', [55].Peso_Real := 593.0, [55].Peso_Teorico := 585.0, [55].No_Cajas := 56, [55].Consec := 107, [55].Envase := 900, [55].Envases_x_Caja := 12, [55].Densidad_Medida := 0.9152, [55].Linea := 1, [56].Fecha.year := 2021, [56].Fecha.Mes := 5, [56].Fecha.Dia := 28, [56].Fecha.Hora := 14, [56].Fecha.Minuto := 42, [56].Fecha.Segundo := 25, [56].Fecha.Milisegundos := 529661, [56].Lote := 148, [56].Operador := 5, [56].Descripcion := 'Alegria Caja 12 x 900 cm3  - Costa', [56].EAN14 := '17702161409646', [56].QAD := '600620', [56].Peso_Real := 548.0, [56].Peso_Teorico := 543.0, [56].No_Cajas := 52, [56].Consec := 109, [56].Envase := 900, [56].Envases_x_Caja := 12, [56].Densidad_Medida := 0.9152, [56].Linea := 1);
   Cola_Estacion_2_A : UDT_COLA[100] := ([0].Fecha.year := 2021, [0].Fecha.Mes := 5, [0].Fecha.Dia := 27, [0].Fecha.Hora := 9, [0].Fecha.Minuto := 12, [0].Fecha.Segundo := 41, [0].Fecha.Milisegundos := 657020, [0].Lote := 147, [0].Operador := 5, [0].Descripcion := 'Alegria Caja 12 x 900 cm3  - Costa', [0].EAN14 := '17702161409646', [0].QAD := '600620', [0].Peso_Real := 595.0, [0].Peso_Teorico := 585.0, [0].No_Cajas := 56, [0].Consec := 13, [0].Envase := 900, [0].Envases_x_Caja := 12, [0].Densidad_Medida := 0.9152, [0].Linea := 1, [1].Fecha.year := 2021, [1].Fecha.Mes := 5, [1].Fecha.Dia := 27, [1].Fecha.Hora := 9, [1].Fecha.Minuto := 25, [1].Fecha.Segundo := 2, [1].Fecha.Milisegundos := 808400, [1].Lote := 147, [1].Operador := 5, [1].Descripcion := 'Alegria Caja 12 x 900 cm3  - Costa', [1].EAN14 := '17702161409646', [1].QAD := '600620', [1].Peso_Real := 596.0, [1].Peso_Teorico := 585.0, [1].No_Cajas := 56, [1].Consec := 17, [1].Envase := 900, [1].Envases_x_Caja := 12, [1].Densidad_Medida := 0.9152, [1].Linea := 1, [2].Fecha.year := 2021, [2].Fecha.Mes := 5, [2].Fecha.Dia := 27, [2].Fecha.Hora := 9, [2].Fecha.Minuto := 29, [2].Fecha.Segundo := 49, [2].Fecha.Milisegundos := 907422, [2].Lote := 147, [2].Operador := 5, [2].Descripcion := 'Alegria Caja 12 x 900 cm3  - Costa', [2].EAN14 := '17702161409646', [2].QAD := '600620', [2].Peso_Real := 595.0, [2].Peso_Teorico := 585.0, [2].No_Cajas := 56, [2].Consec := 19, [2].Envase := 900, [2].Envases_x_Caja := 12, [2].Densidad_Medida := 0.9152, [2].Linea := 1,
        [3].Fecha.year := 2021, [3].Fecha.Mes := 5, [3].Fecha.Dia := 27, [3].Fecha.Hora := 9, [3].Fecha.Minuto := 46, [3].Fecha.Segundo := 24, [3].Fecha.Milisegundos := 347416, [3].Lote := 147, [3].Operador := 5, [3].Descripcion := 'Alegria Caja 12 x 900 cm3  - Costa', [3].EAN14 := '17702161409646', [3].QAD := '600620', [3].Peso_Real := 316.0, [3].Peso_Teorico := 314.0, [3].No_Cajas := 30, [3].Consec := 23, [3].Envase := 900, [3].Envases_x_Caja := 12, [3].Densidad_Medida := 0.9152, [3].Linea := 1, [4].Fecha.year := 2021, [4].Fecha.Mes := 5, [4].Fecha.Dia := 27, [4].Fecha.Hora := 9, [4].Fecha.Minuto := 50, [4].Fecha.Segundo := 2, [4].Fecha.Milisegundos := 369934, [4].Lote := 147, [4].Operador := 5, [4].Descripcion := 'Alegria Caja 12 x 900 cm3  - Costa', [4].EAN14 := '17702161409646', [4].QAD := '600620', [4].Peso_Real := 432.0, [4].Peso_Teorico := 428.0, [4].No_Cajas := 41, [4].Consec := 25, [4].Envase := 900, [4].Envases_x_Caja := 12, [4].Densidad_Medida := 0.9152, [4].Linea := 1, [5].Fecha.year := 2021, [5].Fecha.Mes := 5, [5].Fecha.Dia := 27, [5].Fecha.Hora := 10, [5].Fecha.Minuto := 37, [5].Fecha.Segundo := 37, [5].Fecha.Milisegundos := 441359, [5].Lote := 147, [5].Operador := 5, [5].Descripcion := 'Alegria Caja 12 x 900 cm3  - Costa', [5].EAN14 := '17702161409646', [5].QAD := '600620', [5].Peso_Real := 589.0, [5].Peso_Teorico := 585.0, [5].No_Cajas := 56, [5].Consec := 32, [5].Envase := 900, [5].Envases_x_Caja := 12, [5].Densidad_Medida := 0.9152, [5].Linea := 1,
        [6].Fecha.year := 2021, [6].Fecha.Mes := 5, [6].Fecha.Dia := 27, [6].Fecha.Hora := 10, [6].Fecha.Minuto := 40, [6].Fecha.Segundo := 47, [6].Fecha.Milisegundos := 960363, [6].Lote := 147, [6].Operador := 5, [6].Descripcion := 'Alegria Caja 12 x 900 cm3  - Costa', [6].EAN14 := '17702161409646', [6].QAD := '600620', [6].Peso_Real := 588.0, [6].Peso_Teorico := 585.0, [6].No_Cajas := 56, [6].Consec := 33, [6].Envase := 900, [6].Envases_x_Caja := 12, [6].Densidad_Medida := 0.9152, [6].Linea := 1, [7].Fecha.year := 2021, [7].Fecha.Mes := 5, [7].Fecha.Dia := 27, [7].Fecha.Hora := 10, [7].Fecha.Minuto := 45, [7].Fecha.Segundo := 4, [7].Fecha.Milisegundos := 521191, [7].Lote := 147, [7].Operador := 5, [7].Descripcion := 'Alegria Caja 12 x 900 cm3  - Costa', [7].EAN14 := '17702161409646', [7].QAD := '600620', [7].Peso_Real := 587.0, [7].Peso_Teorico := 585.0, [7].No_Cajas := 56, [7].Consec := 34, [7].Envase := 900, [7].Envases_x_Caja := 12, [7].Densidad_Medida := 0.9152, [7].Linea := 1, [8].Fecha.year := 2021, [8].Fecha.Mes := 5, [8].Fecha.Dia := 27, [8].Fecha.Hora := 10, [8].Fecha.Minuto := 49, [8].Fecha.Segundo := 20, [8].Fecha.Milisegundos := 99146, [8].Lote := 147, [8].Operador := 5, [8].Descripcion := 'Alegria Caja 12 x 900 cm3  - Costa', [8].EAN14 := '17702161409646', [8].QAD := '600620', [8].Peso_Real := 588.0, [8].Peso_Teorico := 585.0, [8].No_Cajas := 56, [8].Consec := 35, [8].Envase := 900, [8].Envases_x_Caja := 12, [8].Densidad_Medida := 0.9152, [8].Linea := 1,
        [9].Fecha.year := 2021, [9].Fecha.Mes := 5, [9].Fecha.Dia := 27, [9].Fecha.Hora := 10, [9].Fecha.Minuto := 50, [9].Fecha.Segundo := 14, [9].Fecha.Milisegundos := 40382, [9].Lote := 147, [9].Operador := 5, [9].Descripcion := 'Alegria Caja 12 x 900 cm3  - Costa', [9].EAN14 := '17702161409646', [9].QAD := '600620', [9].Peso_Real := 574.0, [9].Peso_Teorico := 585.0, [9].No_Cajas := 56, [9].Consec := 36, [9].Envase := 900, [9].Envases_x_Caja := 12, [9].Densidad_Medida := 0.9152, [9].Linea := 1, [10].Fecha.year := 2021, [10].Fecha.Mes := 5, [10].Fecha.Dia := 27, [10].Fecha.Hora := 10, [10].Fecha.Minuto := 52, [10].Fecha.Segundo := 13, [10].Fecha.Milisegundos := 222663, [10].Lote := 147, [10].Operador := 5, [10].Descripcion := 'Alegria Caja 12 x 900 cm3  - Costa', [10].EAN14 := '17702161409646', [10].QAD := '600620', [10].Peso_Real := 589.0, [10].Peso_Teorico := 585.0, [10].No_Cajas := 56, [10].Consec := 37, [10].Envase := 900, [10].Envases_x_Caja := 12, [10].Densidad_Medida := 0.9152, [10].Linea := 1, [11].Fecha.year := 2021, [11].Fecha.Mes := 5, [11].Fecha.Dia := 27, [11].Fecha.Hora := 10, [11].Fecha.Minuto := 52, [11].Fecha.Segundo := 36, [11].Fecha.Milisegundos := 840530, [11].Lote := 147, [11].Operador := 5, [11].Descripcion := 'Alegria Caja 12 x 900 cm3  - Costa', [11].EAN14 := '17702161409646', [11].QAD := '600620', [11].Peso_Real := 588.0, [11].Peso_Teorico := 585.0, [11].No_Cajas := 56, [11].Consec := 38, [11].Envase := 900, [11].Envases_x_Caja := 12, [11].Densidad_Medida := 0.9152, [11].Linea := 1,
        [12].Fecha.year := 2021, [12].Fecha.Mes := 5, [12].Fecha.Dia := 27, [12].Fecha.Hora := 11, [12].Fecha.Minuto := 22, [12].Fecha.Segundo := 51, [12].Fecha.Milisegundos := 758089, [12].Lote := 147, [12].Operador := 5, [12].Descripcion := 'Alegria Caja 12 x 900 cm3  - Costa', [12].EAN14 := '17702161409646', [12].QAD := '600620', [12].Peso_Real := 589.0, [12].Peso_Teorico := 585.0, [12].No_Cajas := 56, [12].Consec := 40, [12].Envase := 900, [12].Envases_x_Caja := 12, [12].Densidad_Medida := 0.9152, [12].Linea := 1, [13].Fecha.year := 2021, [13].Fecha.Mes := 5, [13].Fecha.Dia := 27, [13].Fecha.Hora := 11, [13].Fecha.Minuto := 33, [13].Fecha.Segundo := 34, [13].Fecha.Milisegundos := 529217, [13].Lote := 147, [13].Operador := 5, [13].Descripcion := 'Alegria Caja 12 x 900 cm3  - Costa', [13].EAN14 := '17702161409646', [13].QAD := '600620', [13].Peso_Real := 588.0, [13].Peso_Teorico := 585.0, [13].No_Cajas := 56, [13].Consec := 42, [13].Envase := 900, [13].Envases_x_Caja := 12, [13].Densidad_Medida := 0.9152, [13].Linea := 1, [14].Fecha.year := 2021, [14].Fecha.Mes := 5, [14].Fecha.Dia := 27, [14].Fecha.Hora := 11, [14].Fecha.Minuto := 37, [14].Fecha.Segundo := 10, [14].Fecha.Milisegundos := 664906, [14].Lote := 147, [14].Operador := 5, [14].Descripcion := 'Alegria Caja 12 x 900 cm3  - Costa', [14].EAN14 := '17702161409646', [14].QAD := '600620', [14].Peso_Real := 589.0, [14].Peso_Teorico := 585.0, [14].No_Cajas := 56, [14].Consec := 44, [14].Envase := 900, [14].Envases_x_Caja := 12, [14].Densidad_Medida := 0.9152, [14].Linea := 1,
        [15].Fecha.year := 2021, [15].Fecha.Mes := 5, [15].Fecha.Dia := 27, [15].Fecha.Hora := 11, [15].Fecha.Minuto := 40, [15].Fecha.Segundo := 1, [15].Fecha.Milisegundos := 257737, [15].Lote := 147, [15].Operador := 5, [15].Descripcion := 'Alegria Caja 12 x 900 cm3  - Costa', [15].EAN14 := '17702161409646', [15].QAD := '600620', [15].Peso_Real := 588.0, [15].Peso_Teorico := 585.0, [15].No_Cajas := 56, [15].Consec := 45, [15].Envase := 900, [15].Envases_x_Caja := 12, [15].Densidad_Medida := 0.9152, [15].Linea := 1, [16].Fecha.year := 2021, [16].Fecha.Mes := 5, [16].Fecha.Dia := 27, [16].Fecha.Hora := 11, [16].Fecha.Minuto := 44, [16].Fecha.Segundo := 46, [16].Fecha.Milisegundos := 989670, [16].Lote := 147, [16].Operador := 5, [16].Descripcion := 'Alegria Caja 12 x 900 cm3  - Costa', [16].EAN14 := '17702161409646', [16].QAD := '600620', [16].Peso_Real := 588.0, [16].Peso_Teorico := 585.0, [16].No_Cajas := 56, [16].Consec := 47, [16].Envase := 900, [16].Envases_x_Caja := 12, [16].Densidad_Medida := 0.9152, [16].Linea := 1, [17].Fecha.year := 2021, [17].Fecha.Mes := 5, [17].Fecha.Dia := 27, [17].Fecha.Hora := 11, [17].Fecha.Minuto := 46, [17].Fecha.Segundo := 49, [17].Fecha.Milisegundos := 650130, [17].Lote := 147, [17].Operador := 5, [17].Descripcion := 'Alegria Caja 12 x 900 cm3  - Costa', [17].EAN14 := '17702161409646', [17].QAD := '600620', [17].Peso_Real := 588.0, [17].Peso_Teorico := 585.0, [17].No_Cajas := 56, [17].Consec := 48, [17].Envase := 900, [17].Envases_x_Caja := 12, [17].Densidad_Medida := 0.9152, [17].Linea := 1,
        [18].Fecha.year := 2021, [18].Fecha.Mes := 5, [18].Fecha.Dia := 27, [18].Fecha.Hora := 11, [18].Fecha.Minuto := 49, [18].Fecha.Segundo := 54, [18].Fecha.Milisegundos := 404227, [18].Lote := 147, [18].Operador := 5, [18].Descripcion := 'Alegria Caja 12 x 900 cm3  - Costa', [18].EAN14 := '17702161409646', [18].QAD := '600620', [18].Peso_Real := 589.0, [18].Peso_Teorico := 585.0, [18].No_Cajas := 56, [18].Consec := 50, [18].Envase := 900, [18].Envases_x_Caja := 12, [18].Densidad_Medida := 0.9152, [18].Linea := 1, [19].Fecha.year := 2021, [19].Fecha.Mes := 5, [19].Fecha.Dia := 27, [19].Fecha.Hora := 11, [19].Fecha.Minuto := 57, [19].Fecha.Segundo := 37, [19].Fecha.Milisegundos := 319972, [19].Lote := 147, [19].Operador := 5, [19].Descripcion := 'Alegria Caja 12 x 900 cm3  - Costa', [19].EAN14 := '17702161409646', [19].QAD := '600620', [19].Peso_Real := 588.0, [19].Peso_Teorico := 585.0, [19].No_Cajas := 56, [19].Consec := 52, [19].Envase := 900, [19].Envases_x_Caja := 12, [19].Densidad_Medida := 0.9152, [19].Linea := 1, [20].Fecha.year := 2021, [20].Fecha.Mes := 5, [20].Fecha.Dia := 27, [20].Fecha.Hora := 12, [20].Fecha.Minuto := 4, [20].Fecha.Segundo := 32, [20].Fecha.Milisegundos := 298318, [20].Lote := 147, [20].Operador := 5, [20].Descripcion := 'Alegria Caja 12 x 900 cm3  - Costa', [20].EAN14 := '17702161409646', [20].QAD := '600620', [20].Peso_Real := 590.0, [20].Peso_Teorico := 585.0, [20].No_Cajas := 56, [20].Consec := 55, [20].Envase := 900, [20].Envases_x_Caja := 12, [20].Densidad_Medida := 0.9152, [20].Linea := 1,
        [21].Fecha.year := 2021, [21].Fecha.Mes := 5, [21].Fecha.Dia := 27, [21].Fecha.Hora := 12, [21].Fecha.Minuto := 7, [21].Fecha.Segundo := 59, [21].Fecha.Milisegundos := 210350, [21].Lote := 147, [21].Operador := 5, [21].Descripcion := 'Alegria Caja 12 x 900 cm3  - Costa', [21].EAN14 := '17702161409646', [21].QAD := '600620', [21].Peso_Real := 589.0, [21].Peso_Teorico := 585.0, [21].No_Cajas := 56, [21].Consec := 57, [21].Envase := 900, [21].Envases_x_Caja := 12, [21].Densidad_Medida := 0.9152, [21].Linea := 1, [22].Fecha.year := 2021, [22].Fecha.Mes := 5, [22].Fecha.Dia := 27, [22].Fecha.Hora := 12, [22].Fecha.Minuto := 10, [22].Fecha.Segundo := 39, [22].Fecha.Milisegundos := 687896, [22].Lote := 147, [22].Operador := 5, [22].Descripcion := 'Alegria Caja 12 x 900 cm3  - Costa', [22].EAN14 := '17702161409646', [22].QAD := '600620', [22].Peso_Real := 588.0, [22].Peso_Teorico := 585.0, [22].No_Cajas := 56, [22].Consec := 58, [22].Envase := 900, [22].Envases_x_Caja := 12, [22].Densidad_Medida := 0.9152, [22].Linea := 1, [23].Fecha.year := 2021, [23].Fecha.Mes := 5, [23].Fecha.Dia := 27, [23].Fecha.Hora := 12, [23].Fecha.Minuto := 15, [23].Fecha.Segundo := 52, [23].Fecha.Milisegundos := 477604, [23].Lote := 147, [23].Operador := 5, [23].Descripcion := 'Alegria Caja 12 x 900 cm3  - Costa', [23].EAN14 := '17702161409646', [23].QAD := '600620', [23].Peso_Real := 588.0, [23].Peso_Teorico := 585.0, [23].No_Cajas := 56, [23].Consec := 60, [23].Envase := 900, [23].Envases_x_Caja := 12, [23].Densidad_Medida := 0.9152, [23].Linea := 1,
        [24].Fecha.year := 2021, [24].Fecha.Mes := 5, [24].Fecha.Dia := 27, [24].Fecha.Hora := 12, [24].Fecha.Minuto := 19, [24].Fecha.Segundo := 24, [24].Fecha.Milisegundos := 750931, [24].Lote := 147, [24].Operador := 5, [24].Descripcion := 'Alegria Caja 12 x 900 cm3  - Costa', [24].EAN14 := '17702161409646', [24].QAD := '600620', [24].Peso_Real := 584.0, [24].Peso_Teorico := 585.0, [24].No_Cajas := 56, [24].Consec := 62, [24].Envase := 900, [24].Envases_x_Caja := 12, [24].Densidad_Medida := 0.9152, [24].Linea := 1, [25].Fecha.year := 2021, [25].Fecha.Mes := 5, [25].Fecha.Dia := 27, [25].Fecha.Hora := 12, [25].Fecha.Minuto := 23, [25].Fecha.Segundo := 2, [25].Fecha.Milisegundos := 29362, [25].Lote := 147, [25].Operador := 5, [25].Descripcion := 'Alegria Caja 12 x 900 cm3  - Costa', [25].EAN14 := '17702161409646', [25].QAD := '600620', [25].Peso_Real := 589.0, [25].Peso_Teorico := 585.0, [25].No_Cajas := 56, [25].Consec := 64, [25].Envase := 900, [25].Envases_x_Caja := 12, [25].Densidad_Medida := 0.9152, [25].Linea := 1, [26].Fecha.year := 2021, [26].Fecha.Mes := 5, [26].Fecha.Dia := 27, [26].Fecha.Hora := 12, [26].Fecha.Minuto := 31, [26].Fecha.Segundo := 17, [26].Fecha.Milisegundos := 672795, [26].Lote := 147, [26].Operador := 5, [26].Descripcion := 'Alegria Caja 12 x 900 cm3  - Costa', [26].EAN14 := '17702161409646', [26].QAD := '600620', [26].Peso_Real := 589.0, [26].Peso_Teorico := 585.0, [26].No_Cajas := 56, [26].Consec := 68, [26].Envase := 900, [26].Envases_x_Caja := 12, [26].Densidad_Medida := 0.9152, [26].Linea := 1,
        [27].Fecha.year := 2021, [27].Fecha.Mes := 5, [27].Fecha.Dia := 27, [27].Fecha.Hora := 12, [27].Fecha.Minuto := 35, [27].Fecha.Segundo := 21, [27].Fecha.Milisegundos := 566723, [27].Lote := 147, [27].Operador := 5, [27].Descripcion := 'Alegria Caja 12 x 900 cm3  - Costa', [27].EAN14 := '17702161409646', [27].QAD := '600620', [27].Peso_Real := 589.0, [27].Peso_Teorico := 585.0, [27].No_Cajas := 56, [27].Consec := 70, [27].Envase := 900, [27].Envases_x_Caja := 12, [27].Densidad_Medida := 0.9152, [27].Linea := 1, [28].Fecha.year := 2021, [28].Fecha.Mes := 5, [28].Fecha.Dia := 27, [28].Fecha.Hora := 12, [28].Fecha.Minuto := 38, [28].Fecha.Segundo := 26, [28].Fecha.Milisegundos := 797161, [28].Lote := 147, [28].Operador := 5, [28].Descripcion := 'Alegria Caja 12 x 900 cm3  - Costa', [28].EAN14 := '17702161409646', [28].QAD := '600620', [28].Peso_Real := 588.0, [28].Peso_Teorico := 585.0, [28].No_Cajas := 56, [28].Consec := 72, [28].Envase := 900, [28].Envases_x_Caja := 12, [28].Densidad_Medida := 0.9152, [28].Linea := 1, [29].Fecha.year := 2021, [29].Fecha.Mes := 5, [29].Fecha.Dia := 27, [29].Fecha.Hora := 12, [29].Fecha.Minuto := 43, [29].Fecha.Segundo := 39, [29].Fecha.Milisegundos := 889542, [29].Lote := 147, [29].Operador := 5, [29].Descripcion := 'Alegria Caja 12 x 900 cm3  - Costa', [29].EAN14 := '17702161409646', [29].QAD := '600620', [29].Peso_Real := 588.0, [29].Peso_Teorico := 585.0, [29].No_Cajas := 56, [29].Consec := 73, [29].Envase := 900, [29].Envases_x_Caja := 12, [29].Densidad_Medida := 0.9152, [29].Linea := 1,
        [30].Fecha.year := 2021, [30].Fecha.Mes := 5, [30].Fecha.Dia := 27, [30].Fecha.Hora := 12, [30].Fecha.Minuto := 46, [30].Fecha.Segundo := 4, [30].Fecha.Milisegundos := 319007, [30].Lote := 147, [30].Operador := 5, [30].Descripcion := 'Alegria Caja 12 x 900 cm3  - Costa', [30].EAN14 := '17702161409646', [30].QAD := '600620', [30].Peso_Real := 592.0, [30].Peso_Teorico := 585.0, [30].No_Cajas := 56, [30].Consec := 75, [30].Envase := 900, [30].Envases_x_Caja := 12, [30].Densidad_Medida := 0.9152, [30].Linea := 1, [31].Fecha.year := 2021, [31].Fecha.Mes := 5, [31].Fecha.Dia := 27, [31].Fecha.Hora := 12, [31].Fecha.Minuto := 48, [31].Fecha.Segundo := 33, [31].Fecha.Milisegundos := 513703, [31].Lote := 147, [31].Operador := 5, [31].Descripcion := 'Alegria Caja 12 x 900 cm3  - Costa', [31].EAN14 := '17702161409646', [31].QAD := '600620', [31].Peso_Real := 585.0, [31].Peso_Teorico := 585.0, [31].No_Cajas := 56, [31].Consec := 76, [31].Envase := 900, [31].Envases_x_Caja := 12, [31].Densidad_Medida := 0.9152, [31].Linea := 1, [32].Fecha.year := 2021, [32].Fecha.Mes := 5, [32].Fecha.Dia := 27, [32].Fecha.Hora := 12, [32].Fecha.Minuto := 51, [32].Fecha.Segundo := 31, [32].Fecha.Milisegundos := 208225, [32].Lote := 147, [32].Operador := 5, [32].Descripcion := 'Alegria Caja 12 x 900 cm3  - Costa', [32].EAN14 := '17702161409646', [32].QAD := '600620', [32].Peso_Real := 592.0, [32].Peso_Teorico := 585.0, [32].No_Cajas := 56, [32].Consec := 78, [32].Envase := 900, [32].Envases_x_Caja := 12, [32].Densidad_Medida := 0.9152, [32].Linea := 1,
        [33].Fecha.year := 2021, [33].Fecha.Mes := 5, [33].Fecha.Dia := 27, [33].Fecha.Hora := 12, [33].Fecha.Minuto := 53, [33].Fecha.Segundo := 32, [33].Fecha.Milisegundos := 267130, [33].Lote := 147, [33].Operador := 5, [33].Descripcion := 'Alegria Caja 12 x 900 cm3  - Costa', [33].EAN14 := '17702161409646', [33].QAD := '600620', [33].Peso_Real := 586.0, [33].Peso_Teorico := 585.0, [33].No_Cajas := 56, [33].Consec := 79, [33].Envase := 900, [33].Envases_x_Caja := 12, [33].Densidad_Medida := 0.9152, [33].Linea := 1, [34].Fecha.year := 2021, [34].Fecha.Mes := 5, [34].Fecha.Dia := 27, [34].Fecha.Hora := 12, [34].Fecha.Minuto := 56, [34].Fecha.Segundo := 5, [34].Fecha.Milisegundos := 708881, [34].Lote := 147, [34].Operador := 5, [34].Descripcion := 'Alegria Caja 12 x 900 cm3  - Costa', [34].EAN14 := '17702161409646', [34].QAD := '600620', [34].Peso_Real := 590.0, [34].Peso_Teorico := 585.0, [34].No_Cajas := 56, [34].Consec := 81, [34].Envase := 900, [34].Envases_x_Caja := 12, [34].Densidad_Medida := 0.9152, [34].Linea := 1, [35].Fecha.year := 2021, [35].Fecha.Mes := 5, [35].Fecha.Dia := 27, [35].Fecha.Hora := 12, [35].Fecha.Minuto := 59, [35].Fecha.Segundo := 57, [35].Fecha.Milisegundos := 876889, [35].Lote := 147, [35].Operador := 5, [35].Descripcion := 'Alegria Caja 12 x 900 cm3  - Costa', [35].EAN14 := '17702161409646', [35].QAD := '600620', [35].Peso_Real := 586.0, [35].Peso_Teorico := 585.0, [35].No_Cajas := 56, [35].Consec := 83, [35].Envase := 900, [35].Envases_x_Caja := 12, [35].Densidad_Medida := 0.9152, [35].Linea := 1,
        [36].Fecha.year := 2021, [36].Fecha.Mes := 5, [36].Fecha.Dia := 27, [36].Fecha.Hora := 13, [36].Fecha.Minuto := 2, [36].Fecha.Segundo := 36, [36].Fecha.Milisegundos := 492021, [36].Lote := 147, [36].Operador := 5, [36].Descripcion := 'Alegria Caja 12 x 900 cm3  - Costa', [36].EAN14 := '17702161409646', [36].QAD := '600620', [36].Peso_Real := 586.0, [36].Peso_Teorico := 585.0, [36].No_Cajas := 56, [36].Consec := 84, [36].Envase := 900, [36].Envases_x_Caja := 12, [36].Densidad_Medida := 0.9152, [36].Linea := 1, [37].Fecha.year := 2021, [37].Fecha.Mes := 5, [37].Fecha.Dia := 27, [37].Fecha.Hora := 13, [37].Fecha.Minuto := 4, [37].Fecha.Segundo := 56, [37].Fecha.Milisegundos := 723168, [37].Lote := 147, [37].Operador := 5, [37].Descripcion := 'Alegria Caja 12 x 900 cm3  - Costa', [37].EAN14 := '17702161409646', [37].QAD := '600620', [37].Peso_Real := 587.0, [37].Peso_Teorico := 585.0, [37].No_Cajas := 56, [37].Consec := 86, [37].Envase := 900, [37].Envases_x_Caja := 12, [37].Densidad_Medida := 0.9152, [37].Linea := 1, [38].Fecha.year := 2021, [38].Fecha.Mes := 5, [38].Fecha.Dia := 27, [38].Fecha.Hora := 13, [38].Fecha.Minuto := 8, [38].Fecha.Segundo := 6, [38].Fecha.Milisegundos := 271966, [38].Lote := 147, [38].Operador := 5, [38].Descripcion := 'Alegria Caja 12 x 900 cm3  - Costa', [38].EAN14 := '17702161409646', [38].QAD := '600620', [38].Peso_Real := 586.0, [38].Peso_Teorico := 585.0, [38].No_Cajas := 56, [38].Consec := 87, [38].Envase := 900, [38].Envases_x_Caja := 12, [38].Densidad_Medida := 0.9152, [38].Linea := 1,
        [39].Fecha.year := 2021, [39].Fecha.Mes := 5, [39].Fecha.Dia := 27, [39].Fecha.Hora := 13, [39].Fecha.Minuto := 12, [39].Fecha.Segundo := 15, [39].Fecha.Milisegundos := 46350, [39].Lote := 147, [39].Operador := 5, [39].Descripcion := 'Alegria Caja 12 x 900 cm3  - Costa', [39].EAN14 := '17702161409646', [39].QAD := '600620', [39].Peso_Real := 582.0, [39].Peso_Teorico := 585.0, [39].No_Cajas := 56, [39].Consec := 88, [39].Envase := 900, [39].Envases_x_Caja := 12, [39].Densidad_Medida := 0.9152, [39].Linea := 1, [40].Fecha.year := 2021, [40].Fecha.Mes := 5, [40].Fecha.Dia := 27, [40].Fecha.Hora := 13, [40].Fecha.Minuto := 16, [40].Fecha.Segundo := 36, [40].Fecha.Milisegundos := 963798, [40].Lote := 147, [40].Operador := 5, [40].Descripcion := 'Alegria Caja 12 x 900 cm3  - Costa', [40].EAN14 := '17702161409646', [40].QAD := '600620', [40].Peso_Real := 586.0, [40].Peso_Teorico := 585.0, [40].No_Cajas := 56, [40].Consec := 90, [40].Envase := 900, [40].Envases_x_Caja := 12, [40].Densidad_Medida := 0.9152, [40].Linea := 1, [41].Fecha.year := 2021, [41].Fecha.Mes := 5, [41].Fecha.Dia := 27, [41].Fecha.Hora := 13, [41].Fecha.Minuto := 19, [41].Fecha.Segundo := 7, [41].Fecha.Milisegundos := 687613, [41].Lote := 147, [41].Operador := 5, [41].Descripcion := 'Alegria Caja 12 x 900 cm3  - Costa', [41].EAN14 := '17702161409646', [41].QAD := '600620', [41].Peso_Real := 582.0, [41].Peso_Teorico := 585.0, [41].No_Cajas := 56, [41].Consec := 92, [41].Envase := 900, [41].Envases_x_Caja := 12, [41].Densidad_Medida := 0.9152, [41].Linea := 1,
        [42].Fecha.year := 2021, [42].Fecha.Mes := 5, [42].Fecha.Dia := 27, [42].Fecha.Hora := 13, [42].Fecha.Minuto := 21, [42].Fecha.Segundo := 43, [42].Fecha.Milisegundos := 474025, [42].Lote := 147, [42].Operador := 5, [42].Descripcion := 'Alegria Caja 12 x 900 cm3  - Costa', [42].EAN14 := '17702161409646', [42].QAD := '600620', [42].Peso_Real := 583.0, [42].Peso_Teorico := 585.0, [42].No_Cajas := 56, [42].Consec := 94, [42].Envase := 900, [42].Envases_x_Caja := 12, [42].Densidad_Medida := 0.9152, [42].Linea := 1, [43].Fecha.year := 2021, [43].Fecha.Mes := 5, [43].Fecha.Dia := 27, [43].Fecha.Hora := 13, [43].Fecha.Minuto := 24, [43].Fecha.Segundo := 17, [43].Fecha.Milisegundos := 146779, [43].Lote := 147, [43].Operador := 5, [43].Descripcion := 'Alegria Caja 12 x 900 cm3  - Costa', [43].EAN14 := '17702161409646', [43].QAD := '600620', [43].Peso_Real := 586.0, [43].Peso_Teorico := 585.0, [43].No_Cajas := 56, [43].Consec := 95, [43].Envase := 900, [43].Envases_x_Caja := 12, [43].Densidad_Medida := 0.9152, [43].Linea := 1, [44].Fecha.year := 2021, [44].Fecha.Mes := 5, [44].Fecha.Dia := 27, [44].Fecha.Hora := 13, [44].Fecha.Minuto := 26, [44].Fecha.Segundo := 28, [44].Fecha.Milisegundos := 593078, [44].Lote := 147, [44].Operador := 5, [44].Descripcion := 'Alegria Caja 12 x 900 cm3  - Costa', [44].EAN14 := '17702161409646', [44].QAD := '600620', [44].Peso_Real := 586.0, [44].Peso_Teorico := 585.0, [44].No_Cajas := 56, [44].Consec := 97, [44].Envase := 900, [44].Envases_x_Caja := 12, [44].Densidad_Medida := 0.9152, [44].Linea := 1,
        [45].Fecha.year := 2021, [45].Fecha.Mes := 5, [45].Fecha.Dia := 27, [45].Fecha.Hora := 13, [45].Fecha.Minuto := 29, [45].Fecha.Segundo := 36, [45].Fecha.Milisegundos := 763147, [45].Lote := 147, [45].Operador := 5, [45].Descripcion := 'Alegria Caja 12 x 900 cm3  - Costa', [45].EAN14 := '17702161409646', [45].QAD := '600620', [45].Peso_Real := 586.0, [45].Peso_Teorico := 585.0, [45].No_Cajas := 56, [45].Consec := 99, [45].Envase := 900, [45].Envases_x_Caja := 12, [45].Densidad_Medida := 0.9152, [45].Linea := 1, [46].Fecha.year := 2021, [46].Fecha.Mes := 5, [46].Fecha.Dia := 27, [46].Fecha.Hora := 13, [46].Fecha.Minuto := 32, [46].Fecha.Segundo := 25, [46].Fecha.Milisegundos := 292930, [46].Lote := 147, [46].Operador := 5, [46].Descripcion := 'Alegria Caja 12 x 900 cm3  - Costa', [46].EAN14 := '17702161409646', [46].QAD := '600620', [46].Peso_Real := 586.0, [46].Peso_Teorico := 585.0, [46].No_Cajas := 56, [46].Consec := 100, [46].Envase := 900, [46].Envases_x_Caja := 12, [46].Densidad_Medida := 0.9152, [46].Linea := 1, [47].Fecha.year := 2021, [47].Fecha.Mes := 5, [47].Fecha.Dia := 27, [47].Fecha.Hora := 13, [47].Fecha.Minuto := 35, [47].Fecha.Segundo := 23, [47].Fecha.Milisegundos := 752143, [47].Lote := 147, [47].Operador := 5, [47].Descripcion := 'Alegria Caja 12 x 900 cm3  - Costa', [47].EAN14 := '17702161409646', [47].QAD := '600620', [47].Peso_Real := 586.0, [47].Peso_Teorico := 585.0, [47].No_Cajas := 56, [47].Consec := 102, [47].Envase := 900, [47].Envases_x_Caja := 12, [47].Densidad_Medida := 0.9152, [47].Linea := 1,
        [48].Fecha.year := 2021, [48].Fecha.Mes := 5, [48].Fecha.Dia := 27, [48].Fecha.Hora := 13, [48].Fecha.Minuto := 37, [48].Fecha.Segundo := 45, [48].Fecha.Milisegundos := 211126, [48].Lote := 147, [48].Operador := 5, [48].Descripcion := 'Alegria Caja 12 x 900 cm3  - Costa', [48].EAN14 := '17702161409646', [48].QAD := '600620', [48].Peso_Real := 584.0, [48].Peso_Teorico := 585.0, [48].No_Cajas := 56, [48].Consec := 103, [48].Envase := 900, [48].Envases_x_Caja := 12, [48].Densidad_Medida := 0.9152, [48].Linea := 1, [49].Fecha.year := 2021, [49].Fecha.Mes := 5, [49].Fecha.Dia := 27, [49].Fecha.Hora := 13, [49].Fecha.Minuto := 40, [49].Fecha.Segundo := 23, [49].Fecha.Milisegundos := 913085, [49].Lote := 147, [49].Operador := 5, [49].Descripcion := 'Alegria Caja 12 x 900 cm3  - Costa', [49].EAN14 := '17702161409646', [49].QAD := '600620', [49].Peso_Real := 590.0, [49].Peso_Teorico := 585.0, [49].No_Cajas := 56, [49].Consec := 105, [49].Envase := 900, [49].Envases_x_Caja := 12, [49].Densidad_Medida := 0.9152, [49].Linea := 1, [50].Fecha.year := 2021, [50].Fecha.Mes := 5, [50].Fecha.Dia := 27, [50].Fecha.Hora := 13, [50].Fecha.Minuto := 43, [50].Fecha.Milisegundos := 218833, [50].Lote := 147, [50].Operador := 5, [50].Descripcion := 'Alegria Caja 12 x 900 cm3  - Costa', [50].EAN14 := '17702161409646', [50].QAD := '600620', [50].Peso_Real := 588.0, [50].Peso_Teorico := 585.0, [50].No_Cajas := 56, [50].Consec := 106, [50].Envase := 900, [50].Envases_x_Caja := 12, [50].Densidad_Medida := 0.9152, [50].Linea := 1, [51].Fecha.year := 2021,
        [51].Fecha.Mes := 5, [51].Fecha.Dia := 27, [51].Fecha.Hora := 13, [51].Fecha.Minuto := 46, [51].Fecha.Segundo := 25, [51].Fecha.Milisegundos := 761523, [51].Lote := 147, [51].Operador := 5, [51].Descripcion := 'Alegria Caja 12 x 900 cm3  - Costa', [51].EAN14 := '17702161409646', [51].QAD := '600620', [51].Peso_Real := 586.0, [51].Peso_Teorico := 585.0, [51].No_Cajas := 56, [51].Consec := 108, [51].Envase := 900, [51].Envases_x_Caja := 12, [51].Densidad_Medida := 0.9152, [51].Linea := 1, [52].Fecha.year := 2021, [52].Fecha.Mes := 5, [52].Fecha.Dia := 27, [52].Fecha.Hora := 13, [52].Fecha.Minuto := 49, [52].Fecha.Segundo := 8, [52].Fecha.Milisegundos := 960810, [52].Lote := 147, [52].Operador := 5, [52].Descripcion := 'Alegria Caja 12 x 900 cm3  - Costa', [52].EAN14 := '17702161409646', [52].QAD := '600620', [52].Peso_Real := 586.0, [52].Peso_Teorico := 585.0, [52].No_Cajas := 56, [52].Consec := 110, [52].Envase := 900, [52].Envases_x_Caja := 12, [52].Densidad_Medida := 0.9152, [52].Linea := 1, [53].Fecha.year := 2021, [53].Fecha.Mes := 5, [53].Fecha.Dia := 27, [53].Fecha.Hora := 13, [53].Fecha.Minuto := 51, [53].Fecha.Segundo := 46, [53].Fecha.Milisegundos := 184181, [53].Lote := 147, [53].Operador := 5, [53].Descripcion := 'Alegria Caja 12 x 900 cm3  - Costa', [53].EAN14 := '17702161409646', [53].QAD := '600620', [53].Peso_Real := 586.0, [53].Peso_Teorico := 585.0, [53].No_Cajas := 56, [53].Consec := 111, [53].Envase := 900, [53].Envases_x_Caja := 12, [53].Densidad_Medida := 0.9152, [53].Linea := 1, [54].Fecha.year := 2021,
        [54].Fecha.Mes := 5, [54].Fecha.Dia := 27, [54].Fecha.Hora := 13, [54].Fecha.Minuto := 54, [54].Fecha.Segundo := 17, [54].Fecha.Milisegundos := 346367, [54].Lote := 147, [54].Operador := 5, [54].Descripcion := 'Alegria Caja 12 x 900 cm3  - Costa', [54].EAN14 := '17702161409646', [54].QAD := '600620', [54].Peso_Real := 585.0, [54].Peso_Teorico := 585.0, [54].No_Cajas := 56, [54].Consec := 113, [54].Envase := 900, [54].Envases_x_Caja := 12, [54].Densidad_Medida := 0.9152, [54].Linea := 1, [55].Fecha.year := 2021, [55].Fecha.Mes := 5, [55].Fecha.Dia := 27, [55].Fecha.Hora := 13, [55].Fecha.Minuto := 56, [55].Fecha.Segundo := 47, [55].Fecha.Milisegundos := 155702, [55].Lote := 147, [55].Operador := 5, [55].Descripcion := 'Alegria Caja 12 x 900 cm3  - Costa', [55].EAN14 := '17702161409646', [55].QAD := '600620', [55].Peso_Real := 586.0, [55].Peso_Teorico := 585.0, [55].No_Cajas := 56, [55].Consec := 114, [55].Envase := 900, [55].Envases_x_Caja := 12, [55].Densidad_Medida := 0.9152, [55].Linea := 1, [56].Fecha.year := 2021, [56].Fecha.Mes := 5, [56].Fecha.Dia := 27, [56].Fecha.Hora := 13, [56].Fecha.Minuto := 59, [56].Fecha.Segundo := 32, [56].Fecha.Milisegundos := 282652, [56].Lote := 147, [56].Operador := 5, [56].Descripcion := 'Alegria Caja 12 x 900 cm3  - Costa', [56].EAN14 := '17702161409646', [56].QAD := '600620', [56].Peso_Real := 589.0, [56].Peso_Teorico := 585.0, [56].No_Cajas := 56, [56].Consec := 115, [56].Envase := 900, [56].Envases_x_Caja := 12, [56].Densidad_Medida := 0.9152, [56].Linea := 1, [57].Fecha.year := 2021,
        [57].Fecha.Mes := 5, [57].Fecha.Dia := 27, [57].Fecha.Hora := 14, [57].Fecha.Minuto := 1, [57].Fecha.Segundo := 57, [57].Fecha.Milisegundos := 651356, [57].Lote := 147, [57].Operador := 5, [57].Descripcion := 'Alegria Caja 12 x 900 cm3  - Costa', [57].EAN14 := '17702161409646', [57].QAD := '600620', [57].Peso_Real := 585.0, [57].Peso_Teorico := 585.0, [57].No_Cajas := 56, [57].Consec := 117, [57].Envase := 900, [57].Envases_x_Caja := 12, [57].Densidad_Medida := 0.9152, [57].Linea := 1, [58].Fecha.year := 2021, [58].Fecha.Mes := 5, [58].Fecha.Dia := 27, [58].Fecha.Hora := 14, [58].Fecha.Minuto := 7, [58].Fecha.Segundo := 32, [58].Fecha.Milisegundos := 404601, [58].Lote := 147, [58].Operador := 5, [58].Descripcion := 'Alegria Caja 12 x 900 cm3  - Costa', [58].EAN14 := '17702161409646', [58].QAD := '600620', [58].Peso_Real := 588.0, [58].Peso_Teorico := 585.0, [58].No_Cajas := 56, [58].Consec := 119, [58].Envase := 900, [58].Envases_x_Caja := 12, [58].Densidad_Medida := 0.9152, [58].Linea := 1, [59].Fecha.year := 2021, [59].Fecha.Mes := 5, [59].Fecha.Dia := 27, [59].Fecha.Hora := 14, [59].Fecha.Minuto := 14, [59].Fecha.Segundo := 57, [59].Fecha.Milisegundos := 727509, [59].Lote := 147, [59].Operador := 5, [59].Descripcion := 'Alegria Caja 12 x 900 cm3  - Costa', [59].EAN14 := '17702161409646', [59].QAD := '600620', [59].Peso_Real := 586.0, [59].Peso_Teorico := 585.0, [59].No_Cajas := 56, [59].Consec := 121, [59].Envase := 900, [59].Envases_x_Caja := 12, [59].Densidad_Medida := 0.9152, [59].Linea := 1, [60].Fecha.year := 2021,
        [60].Fecha.Mes := 5, [60].Fecha.Dia := 27, [60].Fecha.Hora := 14, [60].Fecha.Minuto := 16, [60].Fecha.Segundo := 5, [60].Fecha.Milisegundos := 973517, [60].Lote := 147, [60].Operador := 5, [60].Descripcion := 'Alegria Caja 12 x 900 cm3  - Costa', [60].EAN14 := '17702161409646', [60].QAD := '600620', [60].Peso_Real := 31.0, [60].Peso_Teorico := 31.0, [60].No_Cajas := 3, [60].Consec := 122, [60].Envase := 900, [60].Envases_x_Caja := 12, [60].Densidad_Medida := 0.9152, [60].Linea := 1, [61].Fecha.year := 2021, [61].Fecha.Mes := 5, [61].Fecha.Dia := 27, [61].Fecha.Hora := 16, [61].Fecha.Minuto := 23, [61].Fecha.Segundo := 9, [61].Fecha.Milisegundos := 219428, [61].Lote := 147, [61].Operador := 5, [61].Descripcion := 'Alegria Caja 12 x 900 cm3  - Costa', [61].EAN14 := '17702161409646', [61].QAD := '600620', [61].Peso_Real := 588.0, [61].Peso_Teorico := 585.0, [61].No_Cajas := 56, [61].Consec := 133, [61].Envase := 900, [61].Envases_x_Caja := 12, [61].Densidad_Medida := 0.9152, [61].Linea := 1);
   Cola_Estacion_3 : UDT_COLA[100];
   Cola_Estacion_3_A : UDT_COLA[100] := ([0].Fecha.year := 2021, [0].Fecha.Mes := 5, [0].Fecha.Dia := 27, [0].Fecha.Hora := 16, [0].Fecha.Minuto := 31, [0].Fecha.Segundo := 6, [0].Fecha.Milisegundos := 727054, [0].Lote := 147, [0].Operador := 5, [0].Descripcion := 'La Muneca Comisariato Caja 6 x 3000 cm3', [0].EAN14 := '11111111111111', [0].QAD := '602800', [0].Peso_Real := 207.0, [0].Peso_Teorico := 207.0, [0].No_Cajas := 12, [0].Consec := 134, [0].Envase := 3000, [0].Envases_x_Caja := 6, [0].Densidad_Medida := 0.9152, [0].Linea := 3, [1].Fecha.year := 2021, [1].Fecha.Mes := 5, [1].Fecha.Dia := 27, [1].Fecha.Hora := 16, [1].Fecha.Minuto := 35, [1].Fecha.Segundo := 54, [1].Fecha.Milisegundos := 573123, [1].Lote := 147, [1].Operador := 5, [1].Descripcion := 'Alegria Caja 6 x 3000 cm3  - Costa', [1].EAN14 := '17702161043987', [1].QAD := '600300', [1].Peso_Real := 516.0, [1].Peso_Teorico := 519.0, [1].No_Cajas := 30, [1].Consec := 135, [1].Envase := 3000, [1].Envases_x_Caja := 6, [1].Densidad_Medida := 0.9152, [1].Linea := 3, [2].Fecha.year := 2021, [2].Fecha.Mes := 5, [2].Fecha.Dia := 27, [2].Fecha.Hora := 16, [2].Fecha.Minuto := 39, [2].Fecha.Segundo := 21, [2].Fecha.Milisegundos := 120807, [2].Lote := 147, [2].Operador := 5, [2].Descripcion := 'Alegria Caja 6 x 3000 cm3  - Costa', [2].EAN14 := '17702161043987', [2].QAD := '600300', [2].Peso_Real := 515.0, [2].Peso_Teorico := 519.0, [2].No_Cajas := 30, [2].Consec := 136, [2].Envase := 3000, [2].Envases_x_Caja := 6, [2].Densidad_Medida := 0.9152, [2].Linea := 3,
        [3].Fecha.year := 2021, [3].Fecha.Mes := 5, [3].Fecha.Dia := 27, [3].Fecha.Hora := 16, [3].Fecha.Minuto := 42, [3].Fecha.Segundo := 31, [3].Fecha.Milisegundos := 577861, [3].Lote := 147, [3].Operador := 5, [3].Descripcion := 'Alegria Caja 6 x 3000 cm3  - Costa', [3].EAN14 := '17702161043987', [3].QAD := '600300', [3].Peso_Real := 517.0, [3].Peso_Teorico := 519.0, [3].No_Cajas := 30, [3].Consec := 137, [3].Envase := 3000, [3].Envases_x_Caja := 6, [3].Densidad_Medida := 0.9152, [3].Linea := 3, [4].Fecha.year := 2021, [4].Fecha.Mes := 5, [4].Fecha.Dia := 27, [4].Fecha.Hora := 16, [4].Fecha.Minuto := 45, [4].Fecha.Segundo := 25, [4].Fecha.Milisegundos := 339428, [4].Lote := 147, [4].Operador := 5, [4].Descripcion := 'Alegria Caja 6 x 3000 cm3  - Costa', [4].EAN14 := '17702161043987', [4].QAD := '600300', [4].Peso_Real := 517.0, [4].Peso_Teorico := 519.0, [4].No_Cajas := 30, [4].Consec := 138, [4].Envase := 3000, [4].Envases_x_Caja := 6, [4].Densidad_Medida := 0.9152, [4].Linea := 3, [5].Fecha.year := 2021, [5].Fecha.Mes := 5, [5].Fecha.Dia := 27, [5].Fecha.Hora := 16, [5].Fecha.Minuto := 48, [5].Fecha.Segundo := 30, [5].Fecha.Milisegundos := 13239, [5].Lote := 147, [5].Operador := 5, [5].Descripcion := 'Alegria Caja 6 x 3000 cm3  - Costa', [5].EAN14 := '17702161043987', [5].QAD := '600300', [5].Peso_Real := 518.0, [5].Peso_Teorico := 519.0, [5].No_Cajas := 30, [5].Consec := 139, [5].Envase := 3000, [5].Envases_x_Caja := 6, [5].Densidad_Medida := 0.9152, [5].Linea := 3,
        [6].Fecha.year := 2021, [6].Fecha.Mes := 5, [6].Fecha.Dia := 27, [6].Fecha.Hora := 16, [6].Fecha.Minuto := 51, [6].Fecha.Segundo := 39, [6].Fecha.Milisegundos := 466244, [6].Lote := 147, [6].Operador := 5, [6].Descripcion := 'Alegria Caja 6 x 3000 cm3  - Costa', [6].EAN14 := '17702161043987', [6].QAD := '600300', [6].Peso_Real := 516.0, [6].Peso_Teorico := 519.0, [6].No_Cajas := 30, [6].Consec := 140, [6].Envase := 3000, [6].Envases_x_Caja := 6, [6].Densidad_Medida := 0.9152, [6].Linea := 3, [7].Fecha.year := 2021, [7].Fecha.Mes := 5, [7].Fecha.Dia := 27, [7].Fecha.Hora := 16, [7].Fecha.Minuto := 54, [7].Fecha.Segundo := 38, [7].Fecha.Milisegundos := 360594, [7].Lote := 147, [7].Operador := 5, [7].Descripcion := 'Alegria Caja 6 x 3000 cm3  - Costa', [7].EAN14 := '17702161043987', [7].QAD := '600300', [7].Peso_Real := 522.0, [7].Peso_Teorico := 519.0, [7].No_Cajas := 30, [7].Consec := 141, [7].Envase := 3000, [7].Envases_x_Caja := 6, [7].Densidad_Medida := 0.9152, [7].Linea := 3, [8].Fecha.year := 2021, [8].Fecha.Mes := 5, [8].Fecha.Dia := 27, [8].Fecha.Hora := 16, [8].Fecha.Minuto := 57, [8].Fecha.Segundo := 41, [8].Fecha.Milisegundos := 709983, [8].Lote := 147, [8].Operador := 5, [8].Descripcion := 'Alegria Caja 6 x 3000 cm3  - Costa', [8].EAN14 := '17702161043987', [8].QAD := '600300', [8].Peso_Real := 522.0, [8].Peso_Teorico := 519.0, [8].No_Cajas := 30, [8].Consec := 142, [8].Envase := 3000, [8].Envases_x_Caja := 6, [8].Densidad_Medida := 0.9152, [8].Linea := 3,
        [9].Fecha.year := 2021, [9].Fecha.Mes := 5, [9].Fecha.Dia := 27, [9].Fecha.Hora := 17, [9].Fecha.Segundo := 50, [9].Fecha.Milisegundos := 898813, [9].Lote := 147, [9].Operador := 5, [9].Descripcion := 'Alegria Caja 6 x 3000 cm3  - Costa', [9].EAN14 := '17702161043987', [9].QAD := '600300', [9].Peso_Real := 518.0, [9].Peso_Teorico := 519.0, [9].No_Cajas := 30, [9].Consec := 143, [9].Envase := 3000, [9].Envases_x_Caja := 6, [9].Densidad_Medida := 0.9152, [9].Linea := 3, [10].Fecha.year := 2021, [10].Fecha.Mes := 5, [10].Fecha.Dia := 27, [10].Fecha.Hora := 17, [10].Fecha.Minuto := 33, [10].Fecha.Segundo := 43, [10].Fecha.Milisegundos := 523752, [10].Lote := 147, [10].Operador := 5, [10].Descripcion := 'Alegria Caja 6 x 3000 cm3  - Costa', [10].EAN14 := '17702161043987', [10].QAD := '600300', [10].Peso_Real := 518.0, [10].Peso_Teorico := 519.0, [10].No_Cajas := 30, [10].Consec := 144, [10].Envase := 3000, [10].Envases_x_Caja := 6, [10].Densidad_Medida := 0.9152, [10].Linea := 3, [11].Fecha.year := 2021, [11].Fecha.Mes := 5, [11].Fecha.Dia := 27, [11].Fecha.Hora := 17, [11].Fecha.Minuto := 41, [11].Fecha.Segundo := 47, [11].Fecha.Milisegundos := 384332, [11].Lote := 147, [11].Operador := 5, [11].Descripcion := 'Alegria Caja 6 x 3000 cm3  - Costa', [11].EAN14 := '17702161043987', [11].QAD := '600300', [11].Peso_Real := 518.0, [11].Peso_Teorico := 519.0, [11].No_Cajas := 30, [11].Consec := 145, [11].Envase := 3000, [11].Envases_x_Caja := 6, [11].Densidad_Medida := 0.9152, [11].Linea := 3, [12].Fecha.year := 2021,
        [12].Fecha.Mes := 5, [12].Fecha.Dia := 27, [12].Fecha.Hora := 17, [12].Fecha.Minuto := 44, [12].Fecha.Segundo := 50, [12].Fecha.Milisegundos := 273394, [12].Lote := 147, [12].Operador := 5, [12].Descripcion := 'Alegria Caja 6 x 3000 cm3  - Costa', [12].EAN14 := '17702161043987', [12].QAD := '600300', [12].Peso_Real := 516.0, [12].Peso_Teorico := 519.0, [12].No_Cajas := 30, [12].Consec := 146, [12].Envase := 3000, [12].Envases_x_Caja := 6, [12].Densidad_Medida := 0.9152, [12].Linea := 3, [13].Fecha.year := 2021, [13].Fecha.Mes := 5, [13].Fecha.Dia := 27, [13].Fecha.Hora := 17, [13].Fecha.Minuto := 47, [13].Fecha.Segundo := 55, [13].Fecha.Milisegundos := 746455, [13].Lote := 147, [13].Operador := 5, [13].Descripcion := 'Alegria Caja 6 x 3000 cm3  - Costa', [13].EAN14 := '17702161043987', [13].QAD := '600300', [13].Peso_Real := 515.0, [13].Peso_Teorico := 519.0, [13].No_Cajas := 30, [13].Consec := 147, [13].Envase := 3000, [13].Envases_x_Caja := 6, [13].Densidad_Medida := 0.9152, [13].Linea := 3, [14].Fecha.year := 2021, [14].Fecha.Mes := 5, [14].Fecha.Dia := 27, [14].Fecha.Hora := 17, [14].Fecha.Minuto := 51, [14].Fecha.Segundo := 9, [14].Fecha.Milisegundos := 685969, [14].Lote := 147, [14].Operador := 5, [14].Descripcion := 'Alegria Caja 6 x 3000 cm3  - Costa', [14].EAN14 := '17702161043987', [14].QAD := '600300', [14].Peso_Real := 515.0, [14].Peso_Teorico := 519.0, [14].No_Cajas := 30, [14].Consec := 148, [14].Envase := 3000, [14].Envases_x_Caja := 6, [14].Densidad_Medida := 0.9152, [14].Linea := 3, [15].Fecha.year := 2021,
        [15].Fecha.Mes := 5, [15].Fecha.Dia := 27, [15].Fecha.Hora := 17, [15].Fecha.Minuto := 54, [15].Fecha.Segundo := 6, [15].Fecha.Milisegundos := 143, [15].Lote := 147, [15].Operador := 5, [15].Descripcion := 'Alegria Caja 6 x 3000 cm3  - Costa', [15].EAN14 := '17702161043987', [15].QAD := '600300', [15].Peso_Real := 516.0, [15].Peso_Teorico := 519.0, [15].No_Cajas := 30, [15].Consec := 149, [15].Envase := 3000, [15].Envases_x_Caja := 6, [15].Densidad_Medida := 0.9152, [15].Linea := 3, [16].Fecha.year := 2021, [16].Fecha.Mes := 5, [16].Fecha.Dia := 27, [16].Fecha.Hora := 17, [16].Fecha.Minuto := 57, [16].Fecha.Segundo := 16, [16].Fecha.Milisegundos := 169578, [16].Lote := 147, [16].Operador := 5, [16].Descripcion := 'Alegria Caja 6 x 3000 cm3  - Costa', [16].EAN14 := '17702161043987', [16].QAD := '600300', [16].Peso_Real := 516.0, [16].Peso_Teorico := 519.0, [16].No_Cajas := 30, [16].Consec := 150, [16].Envase := 3000, [16].Envases_x_Caja := 6, [16].Densidad_Medida := 0.9152, [16].Linea := 3, [17].Fecha.year := 2021, [17].Fecha.Mes := 5, [17].Fecha.Dia := 27, [17].Fecha.Hora := 18, [17].Fecha.Segundo := 14, [17].Fecha.Milisegundos := 683834, [17].Lote := 147, [17].Operador := 5, [17].Descripcion := 'Alegria Caja 6 x 3000 cm3  - Costa', [17].EAN14 := '17702161043987', [17].QAD := '600300', [17].Peso_Real := 515.0, [17].Peso_Teorico := 519.0, [17].No_Cajas := 30, [17].Consec := 151, [17].Envase := 3000, [17].Envases_x_Caja := 6, [17].Densidad_Medida := 0.9152, [17].Linea := 3, [18].Fecha.year := 2021, [18].Fecha.Mes := 5,
        [18].Fecha.Dia := 27, [18].Fecha.Hora := 18, [18].Fecha.Minuto := 3, [18].Fecha.Segundo := 29, [18].Fecha.Milisegundos := 298249, [18].Lote := 147, [18].Operador := 5, [18].Descripcion := 'Alegria Caja 6 x 3000 cm3  - Costa', [18].EAN14 := '17702161043987', [18].QAD := '600300', [18].Peso_Real := 515.0, [18].Peso_Teorico := 519.0, [18].No_Cajas := 30, [18].Consec := 152, [18].Envase := 3000, [18].Envases_x_Caja := 6, [18].Densidad_Medida := 0.9152, [18].Linea := 3, [19].Fecha.year := 2021, [19].Fecha.Mes := 5, [19].Fecha.Dia := 27, [19].Fecha.Hora := 18, [19].Fecha.Minuto := 6, [19].Fecha.Segundo := 37, [19].Fecha.Milisegundos := 632337, [19].Lote := 147, [19].Operador := 5, [19].Descripcion := 'Alegria Caja 6 x 3000 cm3  - Costa', [19].EAN14 := '17702161043987', [19].QAD := '600300', [19].Peso_Real := 515.0, [19].Peso_Teorico := 519.0, [19].No_Cajas := 30, [19].Consec := 153, [19].Envase := 3000, [19].Envases_x_Caja := 6, [19].Densidad_Medida := 0.9152, [19].Linea := 3, [20].Fecha.year := 2021, [20].Fecha.Mes := 5, [20].Fecha.Dia := 27, [20].Fecha.Hora := 18, [20].Fecha.Minuto := 9, [20].Fecha.Segundo := 44, [20].Fecha.Milisegundos := 938788, [20].Lote := 147, [20].Operador := 5, [20].Descripcion := 'Alegria Caja 6 x 3000 cm3  - Costa', [20].EAN14 := '17702161043987', [20].QAD := '600300', [20].Peso_Real := 514.0, [20].Peso_Teorico := 519.0, [20].No_Cajas := 30, [20].Consec := 154, [20].Envase := 3000, [20].Envases_x_Caja := 6, [20].Densidad_Medida := 0.9152, [20].Linea := 3, [21].Fecha.year := 2021, [21].Fecha.Mes := 5,
        [21].Fecha.Dia := 27, [21].Fecha.Hora := 18, [21].Fecha.Minuto := 13, [21].Fecha.Segundo := 53, [21].Fecha.Milisegundos := 581963, [21].Lote := 147, [21].Operador := 5, [21].Descripcion := 'Alegria Caja 6 x 3000 cm3  - Costa', [21].EAN14 := '17702161043987', [21].QAD := '600300', [21].Peso_Real := 516.0, [21].Peso_Teorico := 519.0, [21].No_Cajas := 30, [21].Consec := 155, [21].Envase := 3000, [21].Envases_x_Caja := 6, [21].Densidad_Medida := 0.9152, [21].Linea := 3, [22].Fecha.year := 2021, [22].Fecha.Mes := 5, [22].Fecha.Dia := 27, [22].Fecha.Hora := 18, [22].Fecha.Minuto := 16, [22].Fecha.Segundo := 21, [22].Fecha.Milisegundos := 632278, [22].Lote := 147, [22].Operador := 5, [22].Descripcion := 'Alegria Caja 6 x 3000 cm3  - Costa', [22].EAN14 := '17702161043987', [22].QAD := '600300', [22].Peso_Real := 515.0, [22].Peso_Teorico := 519.0, [22].No_Cajas := 30, [22].Consec := 156, [22].Envase := 3000, [22].Envases_x_Caja := 6, [22].Densidad_Medida := 0.9152, [22].Linea := 3, [23].Fecha.year := 2021, [23].Fecha.Mes := 5, [23].Fecha.Dia := 27, [23].Fecha.Hora := 18, [23].Fecha.Minuto := 19, [23].Fecha.Segundo := 12, [23].Fecha.Milisegundos := 129004, [23].Lote := 147, [23].Operador := 5, [23].Descripcion := 'Alegria Caja 6 x 3000 cm3  - Costa', [23].EAN14 := '17702161043987', [23].QAD := '600300', [23].Peso_Real := 517.0, [23].Peso_Teorico := 519.0, [23].No_Cajas := 30, [23].Consec := 157, [23].Envase := 3000, [23].Envases_x_Caja := 6, [23].Densidad_Medida := 0.9152, [23].Linea := 3, [24].Fecha.year := 2021, [24].Fecha.Mes := 5,
        [24].Fecha.Dia := 27, [24].Fecha.Hora := 18, [24].Fecha.Minuto := 22, [24].Fecha.Segundo := 17, [24].Fecha.Milisegundos := 720679, [24].Lote := 147, [24].Operador := 5, [24].Descripcion := 'Alegria Caja 6 x 3000 cm3  - Costa', [24].EAN14 := '17702161043987', [24].QAD := '600300', [24].Peso_Real := 517.0, [24].Peso_Teorico := 519.0, [24].No_Cajas := 30, [24].Consec := 158, [24].Envase := 3000, [24].Envases_x_Caja := 6, [24].Densidad_Medida := 0.9152, [24].Linea := 3, [25].Fecha.year := 2021, [25].Fecha.Mes := 5, [25].Fecha.Dia := 27, [25].Fecha.Hora := 18, [25].Fecha.Minuto := 25, [25].Fecha.Segundo := 29, [25].Fecha.Milisegundos := 407255, [25].Lote := 147, [25].Operador := 5, [25].Descripcion := 'Alegria Caja 6 x 3000 cm3  - Costa', [25].EAN14 := '17702161043987', [25].QAD := '600300', [25].Peso_Real := 516.0, [25].Peso_Teorico := 519.0, [25].No_Cajas := 30, [25].Consec := 159, [25].Envase := 3000, [25].Envases_x_Caja := 6, [25].Densidad_Medida := 0.9152, [25].Linea := 3, [26].Fecha.year := 2021, [26].Fecha.Mes := 5, [26].Fecha.Dia := 27, [26].Fecha.Hora := 18, [26].Fecha.Minuto := 28, [26].Fecha.Segundo := 24, [26].Fecha.Milisegundos := 708062, [26].Lote := 147, [26].Operador := 5, [26].Descripcion := 'Alegria Caja 6 x 3000 cm3  - Costa', [26].EAN14 := '17702161043987', [26].QAD := '600300', [26].Peso_Real := 517.0, [26].Peso_Teorico := 519.0, [26].No_Cajas := 30, [26].Consec := 160, [26].Envase := 3000, [26].Envases_x_Caja := 6, [26].Densidad_Medida := 0.9152, [26].Linea := 3, [27].Fecha.year := 2021, [27].Fecha.Mes := 5,
        [27].Fecha.Dia := 27, [27].Fecha.Hora := 18, [27].Fecha.Minuto := 31, [27].Fecha.Segundo := 28, [27].Fecha.Milisegundos := 945097, [27].Lote := 147, [27].Operador := 5, [27].Descripcion := 'Alegria Caja 6 x 3000 cm3  - Costa', [27].EAN14 := '17702161043987', [27].QAD := '600300', [27].Peso_Real := 515.0, [27].Peso_Teorico := 519.0, [27].No_Cajas := 30, [27].Consec := 161, [27].Envase := 3000, [27].Envases_x_Caja := 6, [27].Densidad_Medida := 0.9152, [27].Linea := 3, [28].Fecha.year := 2021, [28].Fecha.Mes := 5, [28].Fecha.Dia := 27, [28].Fecha.Hora := 18, [28].Fecha.Minuto := 34, [28].Fecha.Segundo := 31, [28].Fecha.Milisegundos := 392580, [28].Lote := 147, [28].Operador := 5, [28].Descripcion := 'Alegria Caja 6 x 3000 cm3  - Costa', [28].EAN14 := '17702161043987', [28].QAD := '600300', [28].Peso_Real := 514.0, [28].Peso_Teorico := 519.0, [28].No_Cajas := 30, [28].Consec := 162, [28].Envase := 3000, [28].Envases_x_Caja := 6, [28].Densidad_Medida := 0.9152, [28].Linea := 3, [29].Fecha.year := 2021, [29].Fecha.Mes := 5, [29].Fecha.Dia := 27, [29].Fecha.Hora := 18, [29].Fecha.Minuto := 38, [29].Fecha.Segundo := 19, [29].Fecha.Milisegundos := 952725, [29].Lote := 147, [29].Operador := 5, [29].Descripcion := 'Alegria Caja 6 x 3000 cm3  - Costa', [29].EAN14 := '17702161043987', [29].QAD := '600300', [29].Peso_Real := 515.0, [29].Peso_Teorico := 519.0, [29].No_Cajas := 30, [29].Consec := 163, [29].Envase := 3000, [29].Envases_x_Caja := 6, [29].Densidad_Medida := 0.9152, [29].Linea := 3, [30].Fecha.year := 2021, [30].Fecha.Mes := 5,
        [30].Fecha.Dia := 27, [30].Fecha.Hora := 18, [30].Fecha.Minuto := 40, [30].Fecha.Segundo := 56, [30].Fecha.Milisegundos := 570890, [30].Lote := 147, [30].Operador := 5, [30].Descripcion := 'Alegria Caja 6 x 3000 cm3  - Costa', [30].EAN14 := '17702161043987', [30].QAD := '600300', [30].Peso_Real := 517.0, [30].Peso_Teorico := 519.0, [30].No_Cajas := 30, [30].Consec := 164, [30].Envase := 3000, [30].Envases_x_Caja := 6, [30].Densidad_Medida := 0.9152, [30].Linea := 3, [31].Fecha.year := 2021, [31].Fecha.Mes := 5, [31].Fecha.Dia := 27, [31].Fecha.Hora := 18, [31].Fecha.Minuto := 43, [31].Fecha.Segundo := 38, [31].Fecha.Milisegundos := 631402, [31].Lote := 147, [31].Operador := 5, [31].Descripcion := 'Alegria Caja 6 x 3000 cm3  - Costa', [31].EAN14 := '17702161043987', [31].QAD := '600300', [31].Peso_Real := 516.0, [31].Peso_Teorico := 519.0, [31].No_Cajas := 30, [31].Consec := 165, [31].Envase := 3000, [31].Envases_x_Caja := 6, [31].Densidad_Medida := 0.9152, [31].Linea := 3, [32].Fecha.year := 2021, [32].Fecha.Mes := 5, [32].Fecha.Dia := 27, [32].Fecha.Hora := 18, [32].Fecha.Minuto := 46, [32].Fecha.Segundo := 40, [32].Fecha.Milisegundos := 556595, [32].Lote := 147, [32].Operador := 5, [32].Descripcion := 'Alegria Caja 6 x 3000 cm3  - Costa', [32].EAN14 := '17702161043987', [32].QAD := '600300', [32].Peso_Real := 516.0, [32].Peso_Teorico := 519.0, [32].No_Cajas := 30, [32].Consec := 166, [32].Envase := 3000, [32].Envases_x_Caja := 6, [32].Densidad_Medida := 0.9152, [32].Linea := 3, [33].Fecha.year := 2021, [33].Fecha.Mes := 5,
        [33].Fecha.Dia := 27, [33].Fecha.Hora := 18, [33].Fecha.Minuto := 49, [33].Fecha.Segundo := 48, [33].Fecha.Milisegundos := 236343, [33].Lote := 147, [33].Operador := 5, [33].Descripcion := 'Alegria Caja 6 x 3000 cm3  - Costa', [33].EAN14 := '17702161043987', [33].QAD := '600300', [33].Peso_Real := 517.0, [33].Peso_Teorico := 519.0, [33].No_Cajas := 30, [33].Consec := 167, [33].Envase := 3000, [33].Envases_x_Caja := 6, [33].Densidad_Medida := 0.9152, [33].Linea := 3, [34].Fecha.year := 2021, [34].Fecha.Mes := 5, [34].Fecha.Dia := 27, [34].Fecha.Hora := 18, [34].Fecha.Minuto := 52, [34].Fecha.Segundo := 55, [34].Fecha.Milisegundos := 237712, [34].Lote := 147, [34].Operador := 5, [34].Descripcion := 'Alegria Caja 6 x 3000 cm3  - Costa', [34].EAN14 := '17702161043987', [34].QAD := '600300', [34].Peso_Real := 517.0, [34].Peso_Teorico := 519.0, [34].No_Cajas := 30, [34].Consec := 168, [34].Envase := 3000, [34].Envases_x_Caja := 6, [34].Densidad_Medida := 0.9152, [34].Linea := 3, [35].Fecha.year := 2021, [35].Fecha.Mes := 5, [35].Fecha.Dia := 27, [35].Fecha.Hora := 18, [35].Fecha.Minuto := 55, [35].Fecha.Segundo := 53, [35].Fecha.Milisegundos := 932070, [35].Lote := 147, [35].Operador := 5, [35].Descripcion := 'Alegria Caja 6 x 3000 cm3  - Costa', [35].EAN14 := '17702161043987', [35].QAD := '600300', [35].Peso_Real := 515.0, [35].Peso_Teorico := 519.0, [35].No_Cajas := 30, [35].Consec := 169, [35].Envase := 3000, [35].Envases_x_Caja := 6, [35].Densidad_Medida := 0.9152, [35].Linea := 3, [36].Fecha.year := 2021, [36].Fecha.Mes := 5,
        [36].Fecha.Dia := 27, [36].Fecha.Hora := 18, [36].Fecha.Minuto := 59, [36].Fecha.Milisegundos := 189000, [36].Lote := 147, [36].Operador := 5, [36].Descripcion := 'Alegria Caja 6 x 3000 cm3  - Costa', [36].EAN14 := '17702161043987', [36].QAD := '600300', [36].Peso_Real := 515.0, [36].Peso_Teorico := 519.0, [36].No_Cajas := 30, [36].Consec := 170, [36].Envase := 3000, [36].Envases_x_Caja := 6, [36].Densidad_Medida := 0.9152, [36].Linea := 3, [37].Fecha.year := 2021, [37].Fecha.Mes := 5, [37].Fecha.Dia := 27, [37].Fecha.Hora := 19, [37].Fecha.Minuto := 2, [37].Fecha.Segundo := 2, [37].Fecha.Milisegundos := 705244, [37].Lote := 147, [37].Operador := 5, [37].Descripcion := 'Alegria Caja 6 x 3000 cm3  - Costa', [37].EAN14 := '17702161043987', [37].QAD := '600300', [37].Peso_Real := 514.0, [37].Peso_Teorico := 519.0, [37].No_Cajas := 30, [37].Consec := 171, [37].Envase := 3000, [37].Envases_x_Caja := 6, [37].Densidad_Medida := 0.9152, [37].Linea := 3, [38].Fecha.year := 2021, [38].Fecha.Mes := 5, [38].Fecha.Dia := 27, [38].Fecha.Hora := 19, [38].Fecha.Minuto := 5, [38].Fecha.Segundo := 6, [38].Fecha.Milisegundos := 290226, [38].Lote := 147, [38].Operador := 5, [38].Descripcion := 'Alegria Caja 6 x 3000 cm3  - Costa', [38].EAN14 := '17702161043987', [38].QAD := '600300', [38].Peso_Real := 518.0, [38].Peso_Teorico := 519.0, [38].No_Cajas := 30, [38].Consec := 172, [38].Envase := 3000, [38].Envases_x_Caja := 6, [38].Densidad_Medida := 0.9152, [38].Linea := 3, [39].Fecha.year := 2021, [39].Fecha.Mes := 5, [39].Fecha.Dia := 27,
        [39].Fecha.Hora := 19, [39].Fecha.Minuto := 8, [39].Fecha.Segundo := 42, [39].Fecha.Milisegundos := 432619, [39].Lote := 147, [39].Operador := 5, [39].Descripcion := 'Alegria Caja 6 x 3000 cm3  - Costa', [39].EAN14 := '17702161043987', [39].QAD := '600300', [39].Peso_Real := 520.0, [39].Peso_Teorico := 519.0, [39].No_Cajas := 30, [39].Consec := 173, [39].Envase := 3000, [39].Envases_x_Caja := 6, [39].Densidad_Medida := 0.9152, [39].Linea := 3, [40].Fecha.year := 2021, [40].Fecha.Mes := 5, [40].Fecha.Dia := 27, [40].Fecha.Hora := 19, [40].Fecha.Minuto := 12, [40].Fecha.Milisegundos := 911603, [40].Lote := 147, [40].Operador := 5, [40].Descripcion := 'Alegria Caja 6 x 3000 cm3  - Costa', [40].EAN14 := '17702161043987', [40].QAD := '600300', [40].Peso_Real := 517.0, [40].Peso_Teorico := 519.0, [40].No_Cajas := 30, [40].Consec := 174, [40].Envase := 3000, [40].Envases_x_Caja := 6, [40].Densidad_Medida := 0.9152, [40].Linea := 3, [41].Fecha.year := 2021, [41].Fecha.Mes := 5, [41].Fecha.Dia := 27, [41].Fecha.Hora := 19, [41].Fecha.Minuto := 14, [41].Fecha.Segundo := 48, [41].Fecha.Milisegundos := 114108, [41].Lote := 147, [41].Operador := 5, [41].Descripcion := 'Alegria Caja 6 x 3000 cm3  - Costa', [41].EAN14 := '17702161043987', [41].QAD := '600300', [41].Peso_Real := 523.0, [41].Peso_Teorico := 519.0, [41].No_Cajas := 30, [41].Consec := 175, [41].Envase := 3000, [41].Envases_x_Caja := 6, [41].Densidad_Medida := 0.9152, [41].Linea := 3, [42].Fecha.year := 2021, [42].Fecha.Mes := 5, [42].Fecha.Dia := 27, [42].Fecha.Hora := 19,
        [42].Fecha.Minuto := 19, [42].Fecha.Segundo := 22, [42].Fecha.Milisegundos := 376780, [42].Lote := 147, [42].Operador := 5, [42].Descripcion := 'Alegria Caja 6 x 3000 cm3  - Costa', [42].EAN14 := '17702161043987', [42].QAD := '600300', [42].Peso_Real := 517.0, [42].Peso_Teorico := 519.0, [42].No_Cajas := 30, [42].Consec := 176, [42].Envase := 3000, [42].Envases_x_Caja := 6, [42].Densidad_Medida := 0.9152, [42].Linea := 3, [43].Fecha.year := 2021, [43].Fecha.Mes := 5, [43].Fecha.Dia := 27, [43].Fecha.Hora := 19, [43].Fecha.Minuto := 21, [43].Fecha.Segundo := 40, [43].Fecha.Milisegundos := 164684, [43].Lote := 147, [43].Operador := 5, [43].Descripcion := 'Alegria Caja 6 x 3000 cm3  - Costa', [43].EAN14 := '17702161043987', [43].QAD := '600300', [43].Peso_Real := 516.0, [43].Peso_Teorico := 519.0, [43].No_Cajas := 30, [43].Consec := 177, [43].Envase := 3000, [43].Envases_x_Caja := 6, [43].Densidad_Medida := 0.9152, [43].Linea := 3, [44].Fecha.year := 2021, [44].Fecha.Mes := 5, [44].Fecha.Dia := 27, [44].Fecha.Hora := 19, [44].Fecha.Minuto := 24, [44].Fecha.Segundo := 13, [44].Fecha.Milisegundos := 406416, [44].Lote := 147, [44].Operador := 5, [44].Descripcion := 'Alegria Caja 6 x 3000 cm3  - Costa', [44].EAN14 := '17702161043987', [44].QAD := '600300', [44].Peso_Real := 521.0, [44].Peso_Teorico := 519.0, [44].No_Cajas := 30, [44].Consec := 178, [44].Envase := 3000, [44].Envases_x_Caja := 6, [44].Densidad_Medida := 0.9152, [44].Linea := 3, [45].Fecha.year := 2021, [45].Fecha.Mes := 5, [45].Fecha.Dia := 27, [45].Fecha.Hora := 19,
        [45].Fecha.Minuto := 27, [45].Fecha.Segundo := 29, [45].Fecha.Milisegundos := 435758, [45].Lote := 147, [45].Operador := 5, [45].Descripcion := 'Alegria Caja 6 x 3000 cm3  - Costa', [45].EAN14 := '17702161043987', [45].QAD := '600300', [45].Peso_Real := 525.0, [45].Peso_Teorico := 519.0, [45].No_Cajas := 30, [45].Consec := 179, [45].Envase := 3000, [45].Envases_x_Caja := 6, [45].Densidad_Medida := 0.9152, [45].Linea := 3, [46].Fecha.year := 2021, [46].Fecha.Mes := 5, [46].Fecha.Dia := 27, [46].Fecha.Hora := 19, [46].Fecha.Minuto := 30, [46].Fecha.Segundo := 42, [46].Fecha.Milisegundos := 786685, [46].Lote := 147, [46].Operador := 5, [46].Descripcion := 'Alegria Caja 6 x 3000 cm3  - Costa', [46].EAN14 := '17702161043987', [46].QAD := '600300', [46].Peso_Real := 519.0, [46].Peso_Teorico := 519.0, [46].No_Cajas := 30, [46].Consec := 180, [46].Envase := 3000, [46].Envases_x_Caja := 6, [46].Densidad_Medida := 0.9152, [46].Linea := 3, [47].Fecha.year := 2021, [47].Fecha.Mes := 5, [47].Fecha.Dia := 27, [47].Fecha.Hora := 19, [47].Fecha.Minuto := 33, [47].Fecha.Segundo := 12, [47].Fecha.Milisegundos := 831399, [47].Lote := 147, [47].Operador := 5, [47].Descripcion := 'Alegria Caja 6 x 3000 cm3  - Costa', [47].EAN14 := '17702161043987', [47].QAD := '600300', [47].Peso_Real := 532.0, [47].Peso_Teorico := 519.0, [47].No_Cajas := 30, [47].Consec := 181, [47].Envase := 3000, [47].Envases_x_Caja := 6, [47].Densidad_Medida := 0.9152, [47].Linea := 3, [48].Fecha.year := 2021, [48].Fecha.Mes := 5, [48].Fecha.Dia := 27, [48].Fecha.Hora := 19,
        [48].Fecha.Minuto := 36, [48].Fecha.Segundo := 14, [48].Fecha.Milisegundos := 612226, [48].Lote := 147, [48].Operador := 5, [48].Descripcion := 'Alegria Caja 6 x 3000 cm3  - Costa', [48].EAN14 := '17702161043987', [48].QAD := '600300', [48].Peso_Real := 517.0, [48].Peso_Teorico := 519.0, [48].No_Cajas := 30, [48].Consec := 182, [48].Envase := 3000, [48].Envases_x_Caja := 6, [48].Densidad_Medida := 0.9152, [48].Linea := 3, [49].Fecha.year := 2021, [49].Fecha.Mes := 5, [49].Fecha.Dia := 27, [49].Fecha.Hora := 19, [49].Fecha.Minuto := 39, [49].Fecha.Segundo := 4, [49].Fecha.Milisegundos := 205812, [49].Lote := 147, [49].Operador := 5, [49].Descripcion := 'Alegria Caja 6 x 3000 cm3  - Costa', [49].EAN14 := '17702161043987', [49].QAD := '600300', [49].Peso_Real := 518.0, [49].Peso_Teorico := 519.0, [49].No_Cajas := 30, [49].Consec := 183, [49].Envase := 3000, [49].Envases_x_Caja := 6, [49].Densidad_Medida := 0.9152, [49].Linea := 3, [50].Fecha.year := 2021, [50].Fecha.Mes := 5, [50].Fecha.Dia := 27, [50].Fecha.Hora := 19, [50].Fecha.Minuto := 42, [50].Fecha.Segundo := 29, [50].Fecha.Milisegundos := 852187, [50].Lote := 147, [50].Operador := 5, [50].Descripcion := 'Alegria Caja 6 x 3000 cm3  - Costa', [50].EAN14 := '17702161043987', [50].QAD := '600300', [50].Peso_Real := 512.0, [50].Peso_Teorico := 519.0, [50].No_Cajas := 30, [50].Consec := 184, [50].Envase := 3000, [50].Envases_x_Caja := 6, [50].Densidad_Medida := 0.9152, [50].Linea := 3, [51].Fecha.year := 2021, [51].Fecha.Mes := 5, [51].Fecha.Dia := 27, [51].Fecha.Hora := 19,
        [51].Fecha.Minuto := 45, [51].Fecha.Segundo := 23, [51].Fecha.Milisegundos := 880018, [51].Lote := 147, [51].Operador := 5, [51].Descripcion := 'Alegria Caja 6 x 3000 cm3  - Costa', [51].EAN14 := '17702161043987', [51].QAD := '600300', [51].Peso_Real := 516.0, [51].Peso_Teorico := 519.0, [51].No_Cajas := 30, [51].Consec := 185, [51].Envase := 3000, [51].Envases_x_Caja := 6, [51].Densidad_Medida := 0.9152, [51].Linea := 3, [52].Fecha.year := 2021, [52].Fecha.Mes := 5, [52].Fecha.Dia := 27, [52].Fecha.Hora := 19, [52].Fecha.Minuto := 48, [52].Fecha.Segundo := 29, [52].Fecha.Milisegundos := 66442, [52].Lote := 147, [52].Operador := 5, [52].Descripcion := 'Alegria Caja 6 x 3000 cm3  - Costa', [52].EAN14 := '17702161043987', [52].QAD := '600300', [52].Peso_Real := 516.0, [52].Peso_Teorico := 519.0, [52].No_Cajas := 30, [52].Consec := 186, [52].Envase := 3000, [52].Envases_x_Caja := 6, [52].Densidad_Medida := 0.9152, [52].Linea := 3, [53].Fecha.year := 2021, [53].Fecha.Mes := 5, [53].Fecha.Dia := 27, [53].Fecha.Hora := 19, [53].Fecha.Minuto := 51, [53].Fecha.Segundo := 24, [53].Fecha.Milisegundos := 929059, [53].Lote := 147, [53].Operador := 5, [53].Descripcion := 'Alegria Caja 6 x 3000 cm3  - Costa', [53].EAN14 := '17702161043987', [53].QAD := '600300', [53].Peso_Real := 520.0, [53].Peso_Teorico := 519.0, [53].No_Cajas := 30, [53].Consec := 187, [53].Envase := 3000, [53].Envases_x_Caja := 6, [53].Densidad_Medida := 0.9152, [53].Linea := 3, [54].Fecha.year := 2021, [54].Fecha.Mes := 5, [54].Fecha.Dia := 27, [54].Fecha.Hora := 19,
